KUKA KRL program: MyProgram_005().src

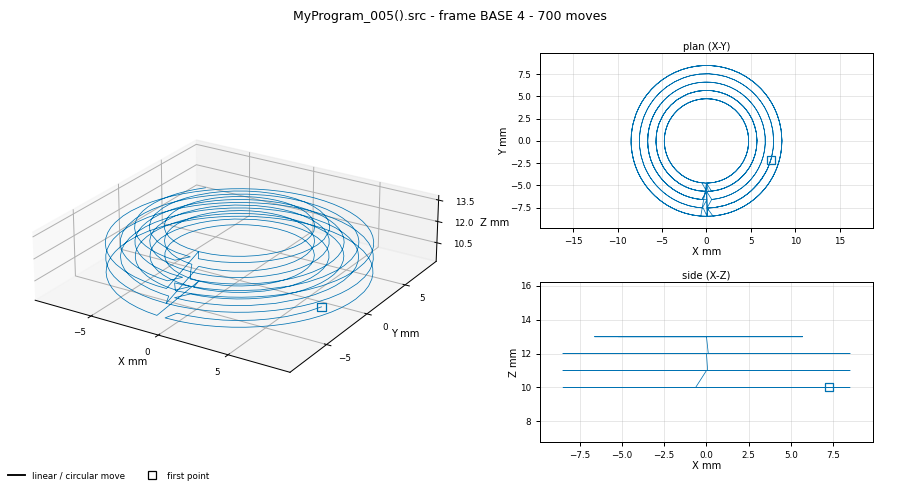
[picture p0: tool path of MyProgram_005().src in frame BASE 4, 700 of 700 moves have a stored position in this frame; points joined in program order, loops and branches not executed]
&ACCESS RVP
&REL 1
&PARAM TEMPLATE = C:\KRC\Roboter\Template\vorgabe
&PARAM EDITMASK = *
DEF MyProgram_005()
; ---- Setting reference (Base) ----
$BASE = BASE_DATA[4]

; --------------------------
; ---- Setting tool (TCP) ----
$TOOL = TOOL_DATA[3]
; --------------------------

$VEL.CP = VEL_APROX_PRINT
Startdeposition()
$VEL.CP = VEL_PRINT
LIN {X 7.2514,Y -2.1135,Z 10,A -2.621,B 0,C 0,E1 0.1598,E2 90.0715} C_DIS
LIN {X 6.8282,Y -3.2375,Z 10,A -2.6842,B 0,C 0,E1 0.1598,E2 90.0713} C_DIS
LIN {X 6.1189,Y -4.4371,Z 10,A -2.7612,B 0,C 0,E1 0.1598,E2 90.0712} C_DIS
LIN {X 5.3653,Y -5.3155,Z 10,A -2.8264,B 0,C 0,E1 0.1598,E2 90.0714} C_DIS
LIN {X 4.7502,Y -5.8723,Z 10,A -2.8729,B 0,C 0,E1 0.1598,E2 90.0716} C_DIS
LIN {X 3.9033,Y -6.4707,Z 10,A -2.9293,B 0,C 0,E1 0.1598,E2 90.0715} C_DIS
LIN {X 3.121,Y -6.8841,Z 10,A -2.9756,B 0,C 0,E1 0.1598,E2 90.0715} C_DIS
LIN {X 2.0664,Y -7.2652,Z 10,A -3.0305,B 0,C 0,E1 0.1598,E2 90.0715} C_DIS
LIN {X 0.9259,Y -7.5003,Z 10,A -3.0823,B 0,C 0,E1 0.1598,E2 90.0715} C_DIS
LIN {X 0.2286,Y -7.5485,Z 10,A -3.11,B 0,C 0,E1 0.1598,E2 90.0715} C_DIS
LIN {X 0.2286,Y -7.5485,Z 10,A -3.11,B 0,C 0,E1 0.1598,E2 90.0715} C_DIS
Enddeposition()
LIN {X -0.0236,Y -8.4916,Z 10,A -3.1582,B 0,C 0,E1 0.1598,E2 90.0702} C_DIS
Startdeposition()
$VEL.CP = VEL_PRINT
LIN {X 0.9995,Y -8.4285,Z 10,A -3.1191,B 0,C 0,E1 0.1598,E2 90.0714} C_DIS
LIN {X 1.8081,Y -8.2918,Z 10,A -3.0837,B 0,C 0,E1 0.1598,E2 90.0714} C_DIS
LIN {X 2.5999,Y -8.0782,Z 10,A -3.0456,B 0,C 0,E1 0.1598,E2 90.0714} C_DIS
LIN {X 3.3672,Y -7.789,Z 10,A -3.0052,B 0,C 0,E1 0.1598,E2 90.0715} C_DIS
LIN {X 4.1031,Y -7.4274,Z 10,A -2.9629,B 0,C 0,E1 0.1598,E2 90.0715} C_DIS
LIN {X 4.8011,Y -6.9971,Z 10,A -2.919,B 0,C 0,E1 0.1598,E2 90.0715} C_DIS
LIN {X 5.4543,Y -6.5014,Z 10,A -2.8739,B 0,C 0,E1 0.1598,E2 90.0716} C_DIS
LIN {X 6.0566,Y -5.9451,Z 10,A -2.8282,B 0,C 0,E1 0.1598,E2 90.0716} C_DIS
LIN {X 6.6023,Y -5.3331,Z 10,A -2.7821,B 0,C 0,E1 0.1598,E2 90.0716} C_DIS
LIN {X 7.0858,Y -4.6709,Z 10,A -2.7362,B 0,C 0,E1 0.1598,E2 90.0716} C_DIS
LIN {X 7.5037,Y -3.9655,Z 10,A -2.6908,B 0,C 0,E1 0.1598,E2 90.0717} C_DIS
LIN {X 7.8515,Y -3.2229,Z 10,A -2.6464,B 0,C 0,E1 0.1598,E2 90.0717} C_DIS
LIN {X 8.1262,Y -2.4503,Z 10,A -2.6035,B 0,C 0,E1 0.1598,E2 90.0717} C_DIS
LIN {X 8.3251,Y -1.6548,Z 10,A -2.5623,B 0,C 0,E1 0.1598,E2 90.0718} C_DIS
LIN {X 8.4456,Y -0.8436,Z 10,A -2.5234,B 0,C 0,E1 0.1598,E2 90.0718} C_DIS
LIN {X 8.4871,Y -0.0246,Z 10,A -2.4871,B 0,C 0,E1 0.1598,E2 90.0718} C_DIS
LIN {X 8.4059,Y 1.2036,Z 10,A -2.4375,B 0,C 0,E1 0.1598,E2 90.0715} C_DIS
LIN {X 8.2317,Y 2.0804,Z 10,A -2.4069,B 0,C 0,E1 0.1598,E2 90.0718} C_DIS
LIN {X 7.9103,Y 3.0772,Z 10,A -2.3765,B 0,C 0,E1 0.1598,E2 90.0718} C_DIS
LIN {X 7.5683,Y 3.8421,Z 10,A -2.3568,B 0,C 0,E1 0.1598,E2 90.0721} C_DIS
LIN {X 7.1528,Y 4.5697,Z 10,A -2.3413,B 0,C 0,E1 0.1598,E2 90.0721} C_DIS
LIN {X 6.6677,Y 5.253,Z 10,A -2.3302,B 0,C 0,E1 0.1598,E2 90.0721} C_DIS
LIN {X 6.1178,Y 5.8852,Z 10,A -2.3238,B 0,C 0,E1 0.1598,E2 90.0722} C_DIS
LIN {X 5.3488,Y 6.5961,Z 10,A -2.3219,B 0,C 0,E1 0.1598,E2 90.0722} C_DIS
LIN {X 4.4236,Y 7.2439,Z 10,A -2.3287,B 0,C 0,E1 0.1598,E2 90.0722} C_DIS
LIN {X 3.6959,Y 7.6405,Z 10,A -2.339,B 0,C 0,E1 0.1598,E2 90.0723} C_DIS
LIN {X 2.9332,Y 7.9646,Z 10,A -2.3535,B 0,C 0,E1 0.1598,E2 90.0723} C_DIS
LIN {X 2.1425,Y 8.213,Z 10,A -2.3722,B 0,C 0,E1 0.1598,E2 90.0723} C_DIS
LIN {X 1.3315,Y 8.3834,Z 10,A -2.395,B 0,C 0,E1 0.1598,E2 90.0723} C_DIS
LIN {X 0.5076,Y 8.4735,Z 10,A -2.4216,B 0,C 0,E1 0.1598,E2 90.0723} C_DIS
LIN {X -0.3211,Y 8.4813,Z 10,A -2.4519,B 0,C 0,E1 0.1598,E2 90.0723} C_DIS
LIN {X -1.1466,Y 8.4087,Z 10,A -2.4855,B 0,C 0,E1 0.1598,E2 90.0723} C_DIS
LIN {X -1.9613,Y 8.2569,Z 10,A -2.522,B 0,C 0,E1 0.1598,E2 90.0723} C_DIS
LIN {X -2.7572,Y 8.026,Z 10,A -2.5611,B 0,C 0,E1 0.1598,E2 90.0721} C_DIS
LIN {X -3.527,Y 7.7188,Z 10,A -2.6024,B 0,C 0,E1 0.1598,E2 90.0721} C_DIS
LIN {X -4.2632,Y 7.3382,Z 10,A -2.6456,B 0,C 0,E1 0.1598,E2 90.072} C_DIS
LIN {X -4.9588,Y 6.8878,Z 10,A -2.6902,B 0,C 0,E1 0.1598,E2 90.0719} C_DIS
LIN {X -5.607,Y 6.3713,Z 10,A -2.7358,B 0,C 0,E1 0.1598,E2 90.0718} C_DIS
LIN {X -6.2028,Y 5.7951,Z 10,A -2.782,B 0,C 0,E1 0.1598,E2 90.0718} C_DIS
LIN {X -6.7386,Y 5.1628,Z 10,A -2.8283,B 0,C 0,E1 0.1598,E2 90.0716} C_DIS
LIN {X -7.2097,Y 4.4809,Z 10,A -2.8743,B 0,C 0,E1 0.1598,E2 90.0716} C_DIS
LIN {X -7.6121,Y 3.7563,Z 10,A -2.9196,B 0,C 0,E1 0.1598,E2 90.0714} C_DIS
LIN {X -7.9422,Y 2.996,Z 10,A -2.9637,B 0,C 0,E1 0.1598,E2 90.0714} C_DIS
LIN {X -8.291,Y 1.8311,Z 10,A -3.0252,B 0,C 0,E1 0.1598,E2 90.0709} C_DIS
LIN {X -8.4593,Y 0.7466,Z 10,A -3.077,B 0,C 0,E1 0.1598,E2 90.0709} C_DIS
LIN {X -8.4789,Y -0.3697,Z 10,A -3.1246,B 0,C 0,E1 0.1598,E2 90.0707} C_DIS
LIN {X -8.4027,Y -1.1872,Z 10,A -3.1566,B 0,C 0,E1 0.1598,E2 90.071} C_DIS
LIN {X -8.2484,Y -1.9937,Z 10,A -3.1848,B 0,C 0,E1 0.1598,E2 90.071} C_DIS
LIN {X -8.0171,Y -2.7815,Z 10,A -3.2095,B 0,C 0,E1 0.1598,E2 90.071} C_DIS
LIN {X -7.7109,Y -3.5434,Z 10,A -3.2304,B 0,C 0,E1 0.1598,E2 90.071} C_DIS
LIN {X -7.3327,Y -4.2722,Z 10,A -3.2472,B 0,C 0,E1 0.1598,E2 90.071} C_DIS
LIN {X -6.8859,Y -4.9612,Z 10,A -3.2599,B 0,C 0,E1 0.1598,E2 90.071} C_DIS
LIN {X -6.3741,Y -5.6034,Z 10,A -3.2682,B 0,C 0,E1 0.1598,E2 90.071} C_DIS
LIN {X -5.8014,Y -6.1919,Z 10,A -3.2721,B 0,C 0,E1 0.1598,E2 90.071} C_DIS
LIN {X -5.176,Y -6.7238,Z 10,A -3.2716,B 0,C 0,E1 0.1598,E2 90.071} C_DIS
LIN {X -4.5041,Y -7.1958,Z 10,A -3.2669,B 0,C 0,E1 0.1598,E2 90.071} C_DIS
LIN {X -3.7871,Y -7.5963,Z 10,A -3.2576,B 0,C 0,E1 0.1598,E2 90.0711} C_DIS
LIN {X -3.0353,Y -7.9267,Z 10,A -3.244,B 0,C 0,E1 0.1598,E2 90.0711} C_DIS
LIN {X -2.2551,Y -8.1827,Z 10,A -3.2263,B 0,C 0,E1 0.1598,E2 90.0712} C_DIS
LIN {X -1.4539,Y -8.3624,Z 10,A -3.2045,B 0,C 0,E1 0.1598,E2 90.0712} C_DIS
LIN {X -0.639,Y -8.4635,Z 10,A -3.179,B 0,C 0,E1 0.1598,E2 90.0713} C_DIS
LIN {X -0.639,Y -8.4635,Z 10,A -3.179,B 0,C 0,E1 0.1598,E2 90.0713} C_DIS
Enddeposition()
LIN {X 0.0003,Y -4.7568,Z 11,A -2.9833,B 0,C 0,E1 0.1598,E2 90.0604} C_DIS
Startdeposition()
$VEL.CP = VEL_PRINT
LIN {X 0.0003,Y -4.7568,Z 11,A -2.9889,B 0,C 0,E1 0.1598,E2 90.0661} C_DIS
LIN {X -0.8726,Y -4.6702,Z 11,A -3.0221,B 0,C 0,E1 0.1598,E2 90.0709} C_DIS
LIN {X -1.5511,Y -4.491,Z 11,A -3.0401,B 0,C 0,E1 0.1598,E2 90.0715} C_DIS
LIN {X -2.1956,Y -4.2133,Z 11,A -3.052,B 0,C 0,E1 0.1598,E2 90.0715} C_DIS
LIN {X -2.7922,Y -3.844,Z 11,A -3.0583,B 0,C 0,E1 0.1598,E2 90.0715} C_DIS
LIN {X -3.3272,Y -3.3898,Z 11,A -3.0587,B 0,C 0,E1 0.1598,E2 90.0714} C_DIS
LIN {X -3.7898,Y -2.8623,Z 11,A -3.0534,B 0,C 0,E1 0.1598,E2 90.0714} C_DIS
LIN {X -4.1709,Y -2.2731,Z 11,A -3.0425,B 0,C 0,E1 0.1598,E2 90.0714} C_DIS
LIN {X -4.4614,Y -1.6344,Z 11,A -3.0262,B 0,C 0,E1 0.1598,E2 90.0714} C_DIS
LIN {X -4.6534,Y -0.9593,Z 11,A -3.0047,B 0,C 0,E1 0.1598,E2 90.0714} C_DIS
LIN {X -4.7423,Y -0.2633,Z 11,A -2.9786,B 0,C 0,E1 0.1598,E2 90.0714} C_DIS
LIN {X -4.731,Y 0.4382,Z 11,A -2.9486,B 0,C 0,E1 0.1598,E2 90.0714} C_DIS
LIN {X -4.6153,Y 1.1305,Z 11,A -2.9152,B 0,C 0,E1 0.1598,E2 90.0714} C_DIS
LIN {X -4.3961,Y 1.7972,Z 11,A -2.879,B 0,C 0,E1 0.1598,E2 90.0715} C_DIS
LIN {X -4.0858,Y 2.4265,Z 11,A -2.8411,B 0,C 0,E1 0.1598,E2 90.0715} C_DIS
LIN {X -3.6841,Y 3.0021,Z 11,A -2.802,B 0,C 0,E1 0.1598,E2 90.0717} C_DIS
LIN {X -3.2012,Y 3.5114,Z 11,A -2.7628,B 0,C 0,E1 0.1598,E2 90.0717} C_DIS
LIN {X -2.6493,Y 3.9451,Z 11,A -2.7242,B 0,C 0,E1 0.1598,E2 90.0719} C_DIS
LIN {X -2.0393,Y 4.2923,Z 11,A -2.6871,B 0,C 0,E1 0.1598,E2 90.0719} C_DIS
LIN {X -1.3842,Y 4.5438,Z 11,A -2.6524,B 0,C 0,E1 0.1598,E2 90.072} C_DIS
LIN {X -0.6998,Y 4.6984,Z 11,A -2.6206,B 0,C 0,E1 0.1598,E2 90.072} C_DIS
LIN {X -0.0003,Y 4.75,Z 11,A -2.5927,B 0,C 0,E1 0.1598,E2 90.0721} C_DIS
LIN {X 0.6994,Y 4.6987,Z 11,A -2.569,B 0,C 0,E1 0.1598,E2 90.0721} C_DIS
LIN {X 1.3838,Y 4.5442,Z 11,A -2.5503,B 0,C 0,E1 0.1598,E2 90.0721} C_DIS
LIN {X 2.039,Y 4.2925,Z 11,A -2.5368,B 0,C 0,E1 0.1598,E2 90.0721} C_DIS
LIN {X 2.6481,Y 3.9439,Z 11,A -2.529,B 0,C 0,E1 0.1598,E2 90.0721} C_DIS
LIN {X 3.1999,Y 3.5104,Z 11,A -2.527,B 0,C 0,E1 0.1598,E2 90.0721} C_DIS
LIN {X 3.6819,Y 3.0005,Z 11,A -2.5308,B 0,C 0,E1 0.1598,E2 90.0721} C_DIS
LIN {X 4.0854,Y 2.4265,Z 11,A -2.5402,B 0,C 0,E1 0.1598,E2 90.072} C_DIS
LIN {X 4.3971,Y 1.7978,Z 11,A -2.5553,B 0,C 0,E1 0.1598,E2 90.072} C_DIS
LIN {X 4.6137,Y 1.1305,Z 11,A -2.5756,B 0,C 0,E1 0.1598,E2 90.0719} C_DIS
LIN {X 4.7302,Y 0.4386,Z 11,A -2.6006,B 0,C 0,E1 0.1598,E2 90.0719} C_DIS
LIN {X 4.7449,Y -0.2631,Z 11,A -2.6298,B 0,C 0,E1 0.1598,E2 90.0718} C_DIS
LIN {X 4.6542,Y -0.959,Z 11,A -2.6627,B 0,C 0,E1 0.1598,E2 90.0718} C_DIS
LIN {X 4.4618,Y -1.634,Z 11,A -2.6984,B 0,C 0,E1 0.1598,E2 90.0718} C_DIS
LIN {X 4.1713,Y -2.2727,Z 11,A -2.7362,B 0,C 0,E1 0.1598,E2 90.0718} C_DIS
LIN {X 3.7907,Y -2.8621,Z 11,A -2.7752,B 0,C 0,E1 0.1598,E2 90.0717} C_DIS
LIN {X 3.2003,Y -3.51,Z 11,A -2.8243,B 0,C 0,E1 0.1598,E2 90.0717} C_DIS
LIN {X 2.648,Y -3.9429,Z 11,A -2.8631,B 0,C 0,E1 0.1598,E2 90.0717} C_DIS
LIN {X 2.1966,Y -4.2139,Z 11,A -2.8912,B 0,C 0,E1 0.1598,E2 90.0717} C_DIS
LIN {X 1.5512,Y -4.4896,Z 11,A -2.9266,B 0,C 0,E1 0.1598,E2 90.0717} C_DIS
LIN {X 0.8732,Y -4.6704,Z 11,A -2.9591,B 0,C 0,E1 0.1598,E2 90.0717} C_DIS
LIN {X 0.0003,Y -4.7568,Z 11,A -2.9948,B 0,C 0,E1 0.1598,E2 90.0716} C_DIS
Enddeposition()
LIN {X 0.0003,Y -4.7568,Z 11,A -2.9948,B 0,C 0,E1 0.1598,E2 90.0716} C_DIS
Startdeposition()
$VEL.CP = VEL_PRINT
LIN {X 0.2115,Y -5.6786,Z 11,A -3.0257,B 0,C 0,E1 0.1598,E2 90.071} C_DIS
LIN {X 1.0414,Y -5.5858,Z 11,A -2.9918,B 0,C 0,E1 0.1598,E2 90.0716} C_DIS
LIN {X 1.849,Y -5.3736,Z 11,A -2.9532,B 0,C 0,E1 0.1598,E2 90.0716} C_DIS
LIN {X 2.6171,Y -5.0456,Z 11,A -2.9111,B 0,C 0,E1 0.1598,E2 90.0716} C_DIS
LIN {X 3.3282,Y -4.6074,Z 11,A -2.8663,B 0,C 0,E1 0.1598,E2 90.0716} C_DIS
LIN {X 4.1901,Y -3.8495,Z 11,A -2.8024,B 0,C 0,E1 0.1598,E2 90.0716} C_DIS
LIN {X 4.8132,Y -3.0255,Z 11,A -2.7445,B 0,C 0,E1 0.1598,E2 90.0716} C_DIS
LIN {X 5.201,Y -2.2955,Z 11,A -2.6993,B 0,C 0,E1 0.1598,E2 90.0716} C_DIS
LIN {X 5.4794,Y -1.5173,Z 11,A -2.656,B 0,C 0,E1 0.1598,E2 90.0717} C_DIS
LIN {X 5.641,Y -0.7067,Z 11,A -2.6156,B 0,C 0,E1 0.1598,E2 90.0717} C_DIS
LIN {X 5.6825,Y 0.1187,Z 11,A -2.579,B 0,C 0,E1 0.1598,E2 90.0717} C_DIS
LIN {X 5.6056,Y 0.9414,Z 11,A -2.547,B 0,C 0,E1 0.1598,E2 90.0718} C_DIS
LIN {X 5.4111,Y 1.7446,Z 11,A -2.5201,B 0,C 0,E1 0.1598,E2 90.0718} C_DIS
LIN {X 5.1013,Y 2.5109,Z 11,A -2.499,B 0,C 0,E1 0.1598,E2 90.0719} C_DIS
LIN {X 4.6827,Y 3.2236,Z 11,A -2.4843,B 0,C 0,E1 0.1598,E2 90.0719} C_DIS
LIN {X 4.165,Y 3.8679,Z 11,A -2.4761,B 0,C 0,E1 0.1598,E2 90.072} C_DIS
LIN {X 3.5608,Y 4.4318,Z 11,A -2.4746,B 0,C 0,E1 0.1598,E2 90.072} C_DIS
LIN {X 2.8804,Y 4.9013,Z 11,A -2.4799,B 0,C 0,E1 0.1598,E2 90.0721} C_DIS
LIN {X 2.1391,Y 5.2669,Z 11,A -2.4918,B 0,C 0,E1 0.1598,E2 90.0721} C_DIS
LIN {X 1.3523,Y 5.5201,Z 11,A -2.5101,B 0,C 0,E1 0.1598,E2 90.0721} C_DIS
LIN {X 0.5378,Y 5.659,Z 11,A -2.5344,B 0,C 0,E1 0.1598,E2 90.0721} C_DIS
LIN {X -0.2883,Y 5.6764,Z 11,A -2.5641,B 0,C 0,E1 0.1598,E2 90.0721} C_DIS
LIN {X -1.1084,Y 5.5748,Z 11,A -2.5986,B 0,C 0,E1 0.1598,E2 90.0721} C_DIS
LIN {X -2.1006,Y 5.2877,Z 11,A -2.6473,B 0,C 0,E1 0.1598,E2 90.072} C_DIS
LIN {X -3.2896,Y 4.6422,Z 11,A -2.7182,B 0,C 0,E1 0.1598,E2 90.0717} C_DIS
LIN {X -3.9903,Y 4.0465,Z 11,A -2.7692,B 0,C 0,E1 0.1598,E2 90.0717} C_DIS
LIN {X -4.4802,Y 3.4976,Z 11,A -2.8104,B 0,C 0,E1 0.1598,E2 90.0717} C_DIS
LIN {X -4.8958,Y 2.8906,Z 11,A -2.8512,B 0,C 0,E1 0.1598,E2 90.0716} C_DIS
LIN {X -5.3507,Y 1.9338,Z 11,A -2.9081,B 0,C 0,E1 0.1598,E2 90.0713} C_DIS
LIN {X -5.5909,Y 1.0258,Z 11,A -2.9552,B 0,C 0,E1 0.1598,E2 90.0713} C_DIS
LIN {X -5.6775,Y 0.2794,Z 11,A -2.9899,B 0,C 0,E1 0.1598,E2 90.0713} C_DIS
LIN {X -5.6649,Y -0.4718,Z 11,A -3.0211,B 0,C 0,E1 0.1598,E2 90.0713} C_DIS
LIN {X -5.5534,Y -1.2149,Z 11,A -3.0484,B 0,C 0,E1 0.1598,E2 90.0713} C_DIS
LIN {X -5.3437,Y -1.9363,Z 11,A -3.0711,B 0,C 0,E1 0.1598,E2 90.0713} C_DIS
LIN {X -5.0406,Y -2.6238,Z 11,A -3.089,B 0,C 0,E1 0.1598,E2 90.0713} C_DIS
LIN {X -4.6521,Y -3.2668,Z 11,A -3.1019,B 0,C 0,E1 0.1598,E2 90.0713} C_DIS
LIN {X -4.1812,Y -3.8525,Z 11,A -3.1093,B 0,C 0,E1 0.1598,E2 90.0713} C_DIS
LIN {X -3.6366,Y -4.3703,Z 11,A -3.1112,B 0,C 0,E1 0.1598,E2 90.0713} C_DIS
LIN {X -3.0273,Y -4.8101,Z 11,A -3.1075,B 0,C 0,E1 0.1598,E2 90.0713} C_DIS
LIN {X -2.3672,Y -5.1692,Z 11,A -3.0985,B 0,C 0,E1 0.1598,E2 90.0713} C_DIS
LIN {X -1.6648,Y -5.4362,Z 11,A -3.084,B 0,C 0,E1 0.1598,E2 90.0714} C_DIS
LIN {X -0.933,Y -5.6073,Z 11,A -3.0644,B 0,C 0,E1 0.1598,E2 90.0714} C_DIS
LIN {X 0.0026,Y -5.6868,Z 11,A -3.0334,B 0,C 0,E1 0.1598,E2 90.0715} C_DIS
Enddeposition()
LIN {X 0.0026,Y -5.6868,Z 11,A -3.0334,B 0,C 0,E1 0.1598,E2 90.0715} C_DIS
Startdeposition()
$VEL.CP = VEL_PRINT
LIN {X -0.4949,Y -6.6014,Z 11,A -3.09,B 0,C 0,E1 0.1598,E2 90.0709} C_DIS
LIN {X -1.1902,Y -6.5105,Z 11,A -3.1122,B 0,C 0,E1 0.1598,E2 90.0714} C_DIS
LIN {X -1.8726,Y -6.3494,Z 11,A -3.1304,B 0,C 0,E1 0.1598,E2 90.0714} C_DIS
LIN {X -2.5337,Y -6.1155,Z 11,A -3.1448,B 0,C 0,E1 0.1598,E2 90.0714} C_DIS
LIN {X -3.1661,Y -5.8125,Z 11,A -3.1552,B 0,C 0,E1 0.1598,E2 90.0714} C_DIS
LIN {X -3.7646,Y -5.4468,Z 11,A -3.1616,B 0,C 0,E1 0.1598,E2 90.0713} C_DIS
LIN {X -4.3185,Y -5.0169,Z 11,A -3.1638,B 0,C 0,E1 0.1598,E2 90.0713} C_DIS
LIN {X -4.8238,Y -4.5307,Z 11,A -3.1618,B 0,C 0,E1 0.1598,E2 90.0713} C_DIS
LIN {X -5.2766,Y -3.9954,Z 11,A -3.1558,B 0,C 0,E1 0.1598,E2 90.0713} C_DIS
LIN {X -5.6699,Y -3.415,Z 11,A -3.1457,B 0,C 0,E1 0.1598,E2 90.0713} C_DIS
LIN {X -5.999,Y -2.7958,Z 11,A -3.1317,B 0,C 0,E1 0.1598,E2 90.0712} C_DIS
LIN {X -6.2622,Y -2.1459,Z 11,A -3.1139,B 0,C 0,E1 0.1598,E2 90.0712} C_DIS
LIN {X -6.4548,Y -1.4716,Z 11,A -3.0926,B 0,C 0,E1 0.1598,E2 90.0712} C_DIS
LIN {X -6.5732,Y -0.7805,Z 11,A -3.0678,B 0,C 0,E1 0.1598,E2 90.0712} C_DIS
LIN {X -6.6178,Y -0.0807,Z 11,A -3.0399,B 0,C 0,E1 0.1598,E2 90.0712} C_DIS
LIN {X -6.5916,Y 0.62,Z 11,A -3.0094,B 0,C 0,E1 0.1598,E2 90.0713} C_DIS
LIN {X -6.4894,Y 1.3139,Z 11,A -2.9765,B 0,C 0,E1 0.1598,E2 90.0713} C_DIS
LIN {X -6.3129,Y 1.9925,Z 11,A -2.9414,B 0,C 0,E1 0.1598,E2 90.0714} C_DIS
LIN {X -6.0681,Y 2.6497,Z 11,A -2.9047,B 0,C 0,E1 0.1598,E2 90.0714} C_DIS
LIN {X -5.7534,Y 3.2763,Z 11,A -2.8667,B 0,C 0,E1 0.1598,E2 90.0716} C_DIS
LIN {X -5.3742,Y 3.8661,Z 11,A -2.8279,B 0,C 0,E1 0.1598,E2 90.0716} C_DIS
LIN {X -4.9335,Y 4.4116,Z 11,A -2.7888,B 0,C 0,E1 0.1598,E2 90.0717} C_DIS
LIN {X -4.4407,Y 4.9103,Z 11,A -2.7496,B 0,C 0,E1 0.1598,E2 90.0717} C_DIS
LIN {X -3.8964,Y 5.3524,Z 11,A -2.7109,B 0,C 0,E1 0.1598,E2 90.0719} C_DIS
LIN {X -3.3078,Y 5.7338,Z 11,A -2.6732,B 0,C 0,E1 0.1598,E2 90.0719} C_DIS
LIN {X -2.6834,Y 6.0528,Z 11,A -2.6367,B 0,C 0,E1 0.1598,E2 90.072} C_DIS
LIN {X -2.0284,Y 6.3032,Z 11,A -2.602,B 0,C 0,E1 0.1598,E2 90.072} C_DIS
LIN {X -1.3505,Y 6.4829,Z 11,A -2.5694,B 0,C 0,E1 0.1598,E2 90.0721} C_DIS
LIN {X -0.6569,Y 6.5864,Z 11,A -2.5395,B 0,C 0,E1 0.1598,E2 90.0721} C_DIS
LIN {X 0.0435,Y 6.6177,Z 11,A -2.5123,B 0,C 0,E1 0.1598,E2 90.0722} C_DIS
LIN {X 0.7435,Y 6.5781,Z 11,A -2.4881,B 0,C 0,E1 0.1598,E2 90.0722} C_DIS
LIN {X 1.4351,Y 6.4616,Z 11,A -2.4675,B 0,C 0,E1 0.1598,E2 90.0722} C_DIS
LIN {X 2.1108,Y 6.2745,Z 11,A -2.4505,B 0,C 0,E1 0.1598,E2 90.0722} C_DIS
LIN {X 2.7627,Y 6.0158,Z 11,A -2.4374,B 0,C 0,E1 0.1598,E2 90.0722} C_DIS
LIN {X 3.3832,Y 5.6892,Z 11,A -2.4283,B 0,C 0,E1 0.1598,E2 90.0722} C_DIS
LIN {X 3.966,Y 5.2993,Z 11,A -2.4232,B 0,C 0,E1 0.1598,E2 90.0722} C_DIS
LIN {X 4.6345,Y 4.7322,Z 11,A -2.4225,B 0,C 0,E1 0.1598,E2 90.0722} C_DIS
LIN {X 5.3297,Y 3.9254,Z 11,A -2.4308,B 0,C 0,E1 0.1598,E2 90.0719} C_DIS
LIN {X 5.7333,Y 3.3083,Z 11,A -2.4423,B 0,C 0,E1 0.1598,E2 90.0721} C_DIS
LIN {X 6.0651,Y 2.65,Z 11,A -2.4579,B 0,C 0,E1 0.1598,E2 90.0721} C_DIS
LIN {X 6.3215,Y 1.9587,Z 11,A -2.4778,B 0,C 0,E1 0.1598,E2 90.072} C_DIS
LIN {X 6.5003,Y 1.2436,Z 11,A -2.5015,B 0,C 0,E1 0.1598,E2 90.072} C_DIS
LIN {X 6.6002,Y 0.513,Z 11,A -2.5288,B 0,C 0,E1 0.1598,E2 90.072} C_DIS
LIN {X 6.6143,Y -0.2241,Z 11,A -2.5596,B 0,C 0,E1 0.1598,E2 90.0719} C_DIS
LIN {X 6.5512,Y -0.9586,Z 11,A -2.5931,B 0,C 0,E1 0.1598,E2 90.0719} C_DIS
LIN {X 6.4028,Y -1.6809,Z 11,A -2.6292,B 0,C 0,E1 0.1598,E2 90.0718} C_DIS
LIN {X 6.1763,Y -2.3825,Z 11,A -2.6673,B 0,C 0,E1 0.1598,E2 90.0718} C_DIS
LIN {X 5.8721,Y -3.0543,Z 11,A -2.707,B 0,C 0,E1 0.1598,E2 90.0718} C_DIS
LIN {X 5.4976,Y -3.6893,Z 11,A -2.7478,B 0,C 0,E1 0.1598,E2 90.0718} C_DIS
LIN {X 5.0529,Y -4.2774,Z 11,A -2.7891,B 0,C 0,E1 0.1598,E2 90.0717} C_DIS
LIN {X 4.5453,Y -4.8123,Z 11,A -2.8305,B 0,C 0,E1 0.1598,E2 90.0717} C_DIS
LIN {X 3.9811,Y -5.287,Z 11,A -2.8714,B 0,C 0,E1 0.1598,E2 90.0717} C_DIS
LIN {X 3.3686,Y -5.6973,Z 11,A -2.9113,B 0,C 0,E1 0.1598,E2 90.0717} C_DIS
LIN {X 2.7135,Y -6.0353,Z 11,A -2.9497,B 0,C 0,E1 0.1598,E2 90.0716} C_DIS
LIN {X 2.0261,Y -6.3017,Z 11,A -2.9862,B 0,C 0,E1 0.1598,E2 90.0716} C_DIS
LIN {X 1.3132,Y -6.49,Z 11,A -3.0204,B 0,C 0,E1 0.1598,E2 90.0716} C_DIS
LIN {X 0.5832,Y -6.5943,Z 11,A -3.0516,B 0,C 0,E1 0.1598,E2 90.0716} C_DIS
LIN {X 0.5832,Y -6.5943,Z 11,A -3.0516,B 0,C 0,E1 0.1598,E2 90.0716} C_DIS
Enddeposition()
LIN {X 0.0612,Y -7.5554,Z 11,A -3.1105,B 0,C 0,E1 0.1598,E2 90.0703} C_DIS
Startdeposition()
$VEL.CP = VEL_PRINT
LIN {X 0.9096,Y -7.5021,Z 11,A -3.0782,B 0,C 0,E1 0.1598,E2 90.0714} C_DIS
LIN {X 2.0698,Y -7.2637,Z 11,A -3.0256,B 0,C 0,E1 0.1598,E2 90.0715} C_DIS
LIN {X 3.159,Y -6.8663,Z 11,A -2.9687,B 0,C 0,E1 0.1598,E2 90.0715} C_DIS
LIN {X 3.97,Y -6.424,Z 11,A -2.9202,B 0,C 0,E1 0.1598,E2 90.0715} C_DIS
LIN {X 4.5787,Y -6.0051,Z 11,A -2.8801,B 0,C 0,E1 0.1598,E2 90.0716} C_DIS
LIN {X 5.6784,Y -4.9864,Z 11,A -2.7959,B 0,C 0,E1 0.1598,E2 90.0712} C_DIS
LIN {X 6.6606,Y -3.5697,Z 11,A -2.6993,B 0,C 0,E1 0.1598,E2 90.071} C_DIS
LIN {X 7.0779,Y -2.6472,Z 11,A -2.6453,B 0,C 0,E1 0.1598,E2 90.0716} C_DIS
LIN {X 7.3848,Y -1.592,Z 11,A -2.589,B 0,C 0,E1 0.1598,E2 90.0716} C_DIS
LIN {X 7.5054,Y -0.8566,Z 11,A -2.5537,B 0,C 0,E1 0.1598,E2 90.0719} C_DIS
LIN {X 7.557,Y 0.0734,Z 11,A -2.512,B 0,C 0,E1 0.1598,E2 90.0717} C_DIS
LIN {X 7.4618,Y 1.1945,Z 11,A -2.4678,B 0,C 0,E1 0.1598,E2 90.0717} C_DIS
LIN {X 7.2396,Y 2.1679,Z 11,A -2.4348,B 0,C 0,E1 0.1598,E2 90.0717} C_DIS
LIN {X 6.907,Y 3.0553,Z 11,A -2.4095,B 0,C 0,E1 0.1598,E2 90.0719} C_DIS
LIN {X 6.5658,Y 3.7322,Z 11,A -2.3935,B 0,C 0,E1 0.1598,E2 90.0721} C_DIS
LIN {X 6.1589,Y 4.3719,Z 11,A -2.3814,B 0,C 0,E1 0.1598,E2 90.0721} C_DIS
LIN {X 5.6894,Y 4.9671,Z 11,A -2.3736,B 0,C 0,E1 0.1598,E2 90.0721} C_DIS
LIN {X 5.1623,Y 5.5119,Z 11,A -2.3699,B 0,C 0,E1 0.1598,E2 90.0722} C_DIS
LIN {X 4.5834,Y 6.0012,Z 11,A -2.3706,B 0,C 0,E1 0.1598,E2 90.0722} C_DIS
LIN {X 3.9597,Y 6.4322,Z 11,A -2.3754,B 0,C 0,E1 0.1598,E2 90.0722} C_DIS
LIN {X 3.1257,Y 6.882,Z 11,A -2.3871,B 0,C 0,E1 0.1598,E2 90.0722} C_DIS
LIN {X 2.194,Y 7.2314,Z 11,A -2.4068,B 0,C 0,E1 0.1598,E2 90.0722} C_DIS
LIN {X 0.9897,Y 7.4881,Z 11,A -2.4405,B 0,C 0,E1 0.1598,E2 90.0722} C_DIS
LIN {X 0.239,Y 7.5535,Z 11,A -2.4655,B 0,C 0,E1 0.1598,E2 90.0722} C_DIS
LIN {X -0.7725,Y 7.5177,Z 11,A -2.5043,B 0,C 0,E1 0.1598,E2 90.0722} C_DIS
LIN {X -1.736,Y 7.3564,Z 11,A -2.5467,B 0,C 0,E1 0.1598,E2 90.0722} C_DIS
LIN {X -2.7886,Y 7.0254,Z 11,A -2.5995,B 0,C 0,E1 0.1598,E2 90.0721} C_DIS
LIN {X -3.6563,Y 6.6078,Z 11,A -2.6491,B 0,C 0,E1 0.1598,E2 90.072} C_DIS
LIN {X -4.4708,Y 6.0944,Z 11,A -2.7007,B 0,C 0,E1 0.1598,E2 90.0718} C_DIS
LIN {X -5.3112,Y 5.37,Z 11,A -2.762,B 0,C 0,E1 0.1598,E2 90.0716} C_DIS
LIN {X -5.8426,Y 4.7877,Z 11,A -2.8062,B 0,C 0,E1 0.1598,E2 90.0716} C_DIS
LIN {X -6.3083,Y 4.1518,Z 11,A -2.8501,B 0,C 0,E1 0.1598,E2 90.0716} C_DIS
LIN {X -6.708,Y 3.4725,Z 11,A -2.8934,B 0,C 0,E1 0.1598,E2 90.0715} C_DIS
LIN {X -7.1059,Y 2.571,Z 11,A -2.9458,B 0,C 0,E1 0.1598,E2 90.0712} C_DIS
LIN {X -7.4227,Y 1.3948,Z 11,A -3.0067,B 0,C 0,E1 0.1598,E2 90.0708} C_DIS
LIN {X -7.5368,Y 0.5156,Z 11,A -3.0482,B 0,C 0,E1 0.1598,E2 90.0711} C_DIS
LIN {X -7.5341,Y -0.5927,Z 11,A -3.0945,B 0,C 0,E1 0.1598,E2 90.0707} C_DIS
LIN {X -7.3917,Y -1.5706,Z 11,A -3.1306,B 0,C 0,E1 0.1598,E2 90.0709} C_DIS
LIN {X -7.0689,Y -2.6624,Z 11,A -3.1646,B 0,C 0,E1 0.1598,E2 90.0707} C_DIS
LIN {X -6.7741,Y -3.3489,Z 11,A -3.183,B 0,C 0,E1 0.1598,E2 90.071} C_DIS
LIN {X -6.2739,Y -4.2128,Z 11,A -3.201,B 0,C 0,E1 0.1598,E2 90.071} C_DIS
LIN {X -5.5619,Y -5.1165,Z 11,A -3.213,B 0,C 0,E1 0.1598,E2 90.0709} C_DIS
LIN {X -4.8434,Y -5.795,Z 11,A -3.2154,B 0,C 0,E1 0.1598,E2 90.0711} C_DIS
LIN {X -4.2115,Y -6.27,Z 11,A -3.2124,B 0,C 0,E1 0.1598,E2 90.0711} C_DIS
LIN {X -3.5333,Y -6.6762,Z 11,A -3.2047,B 0,C 0,E1 0.1598,E2 90.0712} C_DIS
LIN {X -2.8161,Y -7.009,Z 11,A -3.1925,B 0,C 0,E1 0.1598,E2 90.0712} C_DIS
LIN {X -1.8779,Y -7.3197,Z 11,A -3.1713,B 0,C 0,E1 0.1598,E2 90.0712} C_DIS
LIN {X -0.9529,Y -7.4938,Z 11,A -3.1448,B 0,C 0,E1 0.1598,E2 90.0714} C_DIS
LIN {X -0.3743,Y -7.5452,Z 11,A -3.1257,B 0,C 0,E1 0.1598,E2 90.0714} C_DIS
LIN {X -0.3743,Y -7.5452,Z 11,A -3.1257,B 0,C 0,E1 0.1598,E2 90.0714} C_DIS
Enddeposition()
LIN {X 0.0683,Y -8.4871,Z 11,A -3.1485,B 0,C 0,E1 0.1598,E2 90.0702} C_DIS
Startdeposition()
$VEL.CP = VEL_PRINT
LIN {X -0.9758,Y -8.4305,Z 11,A -3.1854,B 0,C 0,E1 0.1598,E2 90.0713} C_DIS
LIN {X -1.8014,Y -8.2948,Z 11,A -3.21,B 0,C 0,E1 0.1598,E2 90.0713} C_DIS
LIN {X -2.6094,Y -8.0774,Z 11,A -3.2304,B 0,C 0,E1 0.1598,E2 90.0713} C_DIS
LIN {X -3.3919,Y -7.781,Z 11,A -3.2465,B 0,C 0,E1 0.1598,E2 90.0712} C_DIS
LIN {X -4.1418,Y -7.4099,Z 11,A -3.2583,B 0,C 0,E1 0.1598,E2 90.0712} C_DIS
LIN {X -4.8515,Y -6.9664,Z 11,A -3.2656,B 0,C 0,E1 0.1598,E2 90.0712} C_DIS
LIN {X -5.5138,Y -6.455,Z 11,A -3.2682,B 0,C 0,E1 0.1598,E2 90.0711} C_DIS
LIN {X -6.1215,Y -5.8798,Z 11,A -3.2662,B 0,C 0,E1 0.1598,E2 90.0711} C_DIS
LIN {X -6.6696,Y -5.2475,Z 11,A -3.2596,B 0,C 0,E1 0.1598,E2 90.0711} C_DIS
LIN {X -7.1551,Y -4.566,Z 11,A -3.2486,B 0,C 0,E1 0.1598,E2 90.071} C_DIS
LIN {X -7.5698,Y -3.8392,Z 11,A -3.2332,B 0,C 0,E1 0.1598,E2 90.071} C_DIS
LIN {X -7.9111,Y -3.0751,Z 11,A -3.2135,B 0,C 0,E1 0.1598,E2 90.071} C_DIS
LIN {X -8.1756,Y -2.2812,Z 11,A -3.1898,B 0,C 0,E1 0.1598,E2 90.071} C_DIS
LIN {X -8.397,Y -1.2589,Z 11,A -3.1546,B 0,C 0,E1 0.1598,E2 90.0707} C_DIS
LIN {X -8.4874,Y -0.2374,Z 11,A -3.115,B 0,C 0,E1 0.1598,E2 90.0709} C_DIS
LIN {X -8.4598,Y 0.7402,Z 11,A -3.0728,B 0,C 0,E1 0.1598,E2 90.0709} C_DIS
LIN {X -8.291,Y 1.8311,Z 11,A -3.0206,B 0,C 0,E1 0.1598,E2 90.0709} C_DIS
LIN {X -7.9448,Y 2.9894,Z 11,A -2.9591,B 0,C 0,E1 0.1598,E2 90.0709} C_DIS
LIN {X -7.6152,Y 3.7501,Z 11,A -2.9153,B 0,C 0,E1 0.1598,E2 90.0714} C_DIS
LIN {X -7.2133,Y 4.4752,Z 11,A -2.87,B 0,C 0,E1 0.1598,E2 90.0714} C_DIS
LIN {X -6.7426,Y 5.1576,Z 11,A -2.824,B 0,C 0,E1 0.1598,E2 90.0716} C_DIS
LIN {X -6.2071,Y 5.7903,Z 11,A -2.7776,B 0,C 0,E1 0.1598,E2 90.0716} C_DIS
LIN {X -5.6121,Y 6.3676,Z 11,A -2.7314,B 0,C 0,E1 0.1598,E2 90.0718} C_DIS
LIN {X -4.9638,Y 6.8842,Z 11,A -2.6858,B 0,C 0,E1 0.1598,E2 90.0718} C_DIS
LIN {X -4.2682,Y 7.3352,Z 11,A -2.6412,B 0,C 0,E1 0.1598,E2 90.072} C_DIS
LIN {X -3.5321,Y 7.7164,Z 11,A -2.598,B 0,C 0,E1 0.1598,E2 90.072} C_DIS
LIN {X -2.7624,Y 8.0241,Z 11,A -2.5566,B 0,C 0,E1 0.1598,E2 90.0721} C_DIS
LIN {X -1.9665,Y 8.2556,Z 11,A -2.5175,B 0,C 0,E1 0.1598,E2 90.0721} C_DIS
LIN {X -1.1517,Y 8.408,Z 11,A -2.481,B 0,C 0,E1 0.1598,E2 90.0723} C_DIS
LIN {X -0.3261,Y 8.481,Z 11,A -2.4474,B 0,C 0,E1 0.1598,E2 90.0723} C_DIS
LIN {X 0.5028,Y 8.4738,Z 11,A -2.4171,B 0,C 0,E1 0.1598,E2 90.0723} C_DIS
LIN {X 1.3269,Y 8.3843,Z 11,A -2.3904,B 0,C 0,E1 0.1598,E2 90.0723} C_DIS
LIN {X 2.1382,Y 8.2143,Z 11,A -2.3676,B 0,C 0,E1 0.1598,E2 90.0723} C_DIS
LIN {X 2.9292,Y 7.9662,Z 11,A -2.3489,B 0,C 0,E1 0.1598,E2 90.0723} C_DIS
LIN {X 3.6923,Y 7.6424,Z 11,A -2.3344,B 0,C 0,E1 0.1598,E2 90.0723} C_DIS
LIN {X 4.4202,Y 7.246,Z 11,A -2.3242,B 0,C 0,E1 0.1598,E2 90.0723} C_DIS
LIN {X 5.345,Y 6.5991,Z 11,A -2.3173,B 0,C 0,E1 0.1598,E2 90.0723} C_DIS
LIN {X 6.1206,Y 5.8817,Z 11,A -2.3191,B 0,C 0,E1 0.1598,E2 90.0722} C_DIS
LIN {X 6.6747,Y 5.2434,Z 11,A -2.3257,B 0,C 0,E1 0.1598,E2 90.0722} C_DIS
LIN {X 7.1626,Y 4.5532,Z 11,A -2.3369,B 0,C 0,E1 0.1598,E2 90.0722} C_DIS
LIN {X 7.5797,Y 3.818,Z 11,A -2.3527,B 0,C 0,E1 0.1598,E2 90.0722} C_DIS
LIN {X 7.9217,Y 3.0451,Z 11,A -2.3729,B 0,C 0,E1 0.1598,E2 90.0721} C_DIS
LIN {X 8.1853,Y 2.242,Z 11,A -2.3972,B 0,C 0,E1 0.1598,E2 90.0721} C_DIS
LIN {X 8.4051,Y 1.2086,Z 11,A -2.4327,B 0,C 0,E1 0.1598,E2 90.0716} C_DIS
LIN {X 8.4904,Y 0.1014,Z 11,A -2.4766,B 0,C 0,E1 0.1598,E2 90.0716} C_DIS
LIN {X 8.4408,Y -0.891,Z 11,A -2.5207,B 0,C 0,E1 0.1598,E2 90.0717} C_DIS
LIN {X 8.3214,Y -1.6769,Z 11,A -2.5587,B 0,C 0,E1 0.1598,E2 90.0718} C_DIS
LIN {X 8.0706,Y -2.6384,Z 11,A -2.6085,B 0,C 0,E1 0.1598,E2 90.0715} C_DIS
LIN {X 7.6152,Y -3.7515,Z 11,A -2.6725,B 0,C 0,E1 0.1598,E2 90.0713} C_DIS
LIN {X 7.2107,Y -4.4808,Z 11,A -2.7187,B 0,C 0,E1 0.1598,E2 90.0717} C_DIS
LIN {X 6.7362,Y -5.1668,Z 11,A -2.7653,B 0,C 0,E1 0.1598,E2 90.0717} C_DIS
LIN {X 6.1963,Y -5.8024,Z 11,A -2.8122,B 0,C 0,E1 0.1598,E2 90.0717} C_DIS
LIN {X 5.5962,Y -6.3816,Z 11,A -2.8588,B 0,C 0,E1 0.1598,E2 90.0716} C_DIS
LIN {X 4.9427,Y -6.8997,Z 11,A -2.9048,B 0,C 0,E1 0.1598,E2 90.0716} C_DIS
LIN {X 4.2415,Y -7.3512,Z 11,A -2.9498,B 0,C 0,E1 0.1598,E2 90.0716} C_DIS
LIN {X 3.4995,Y -7.7318,Z 11,A -2.9931,B 0,C 0,E1 0.1598,E2 90.0716} C_DIS
LIN {X 2.7238,Y -8.0379,Z 11,A -3.0346,B 0,C 0,E1 0.1598,E2 90.0715} C_DIS
LIN {X 1.9218,Y -8.2665,Z 11,A -3.0737,B 0,C 0,E1 0.1598,E2 90.0715} C_DIS
LIN {X 0.8946,Y -8.4434,Z 11,A -3.1189,B 0,C 0,E1 0.1598,E2 90.0715} C_DIS
LIN {X 0.0683,Y -8.4871,Z 11,A -3.151,B 0,C 0,E1 0.1598,E2 90.0714} C_DIS
Enddeposition()
LIN {X 0.0003,Y -4.7568,Z 12,A -2.9802,B 0,C 0,E1 0.1598,E2 90.0604} C_DIS
Startdeposition()
$VEL.CP = VEL_PRINT
LIN {X 0.0003,Y -4.7568,Z 12,A -2.9859,B 0,C 0,E1 0.1598,E2 90.0661} C_DIS
LIN {X 0.8632,Y -4.6726,Z 12,A -2.9555,B 0,C 0,E1 0.1598,E2 90.071} C_DIS
LIN {X 1.6156,Y -4.4663,Z 12,A -2.9197,B 0,C 0,E1 0.1598,E2 90.0716} C_DIS
LIN {X 2.1728,Y -4.2257,Z 12,A -2.8891,B 0,C 0,E1 0.1598,E2 90.0716} C_DIS
LIN {X 2.8338,Y -3.8114,Z 12,A -2.8472,B 0,C 0,E1 0.1598,E2 90.0716} C_DIS
LIN {X 3.2982,Y -3.4206,Z 12,A -2.8136,B 0,C 0,E1 0.1598,E2 90.0717} C_DIS
LIN {X 3.7598,Y -2.9029,Z 12,A -2.7746,B 0,C 0,E1 0.1598,E2 90.0717} C_DIS
LIN {X 4.1427,Y -2.3247,Z 12,A -2.736,B 0,C 0,E1 0.1598,E2 90.0717} C_DIS
LIN {X 4.4369,Y -1.6968,Z 12,A -2.6985,B 0,C 0,E1 0.1598,E2 90.0717} C_DIS
LIN {X 4.6369,Y -1.0327,Z 12,A -2.6629,B 0,C 0,E1 0.1598,E2 90.0717} C_DIS
LIN {X 4.7377,Y -0.3466,Z 12,A -2.6301,B 0,C 0,E1 0.1598,E2 90.0718} C_DIS
LIN {X 4.738,Y 0.3469,Z 12,A -2.6007,B 0,C 0,E1 0.1598,E2 90.0718} C_DIS
LIN {X 4.6365,Y 1.0329,Z 12,A -2.5753,B 0,C 0,E1 0.1598,E2 90.0718} C_DIS
LIN {X 4.4366,Y 1.697,Z 12,A -2.5546,B 0,C 0,E1 0.1598,E2 90.0719} C_DIS
LIN {X 4.1427,Y 2.325,Z 12,A -2.5388,B 0,C 0,E1 0.1598,E2 90.0719} C_DIS
LIN {X 3.7594,Y 2.9029,Z 12,A -2.5285,B 0,C 0,E1 0.1598,E2 90.072} C_DIS
LIN {X 3.2963,Y 3.419,Z 12,A -2.5237,B 0,C 0,E1 0.1598,E2 90.072} C_DIS
LIN {X 2.7649,Y 3.8648,Z 12,A -2.5245,B 0,C 0,E1 0.1598,E2 90.072} C_DIS
LIN {X 2.1719,Y 4.2247,Z 12,A -2.5311,B 0,C 0,E1 0.1598,E2 90.0721} C_DIS
LIN {X 1.5333,Y 4.495,Z 12,A -2.5433,B 0,C 0,E1 0.1598,E2 90.0721} C_DIS
LIN {X 0.8625,Y 4.671,Z 12,A -2.5606,B 0,C 0,E1 0.1598,E2 90.0721} C_DIS
LIN {X 0.1733,Y 4.7492,Z 12,A -2.5827,B 0,C 0,E1 0.1598,E2 90.0721} C_DIS
LIN {X -0.5199,Y 4.7233,Z 12,A -2.6094,B 0,C 0,E1 0.1598,E2 90.0721} C_DIS
LIN {X -1.202,Y 4.5969,Z 12,A -2.6399,B 0,C 0,E1 0.1598,E2 90.0721} C_DIS
LIN {X -1.8586,Y 4.3733,Z 12,A -2.6735,B 0,C 0,E1 0.1598,E2 90.072} C_DIS
LIN {X -2.4744,Y 4.0544,Z 12,A -2.7096,B 0,C 0,E1 0.1598,E2 90.072} C_DIS
LIN {X -3.0385,Y 3.6512,Z 12,A -2.7474,B 0,C 0,E1 0.1598,E2 90.0718} C_DIS
LIN {X -3.5377,Y 3.1698,Z 12,A -2.786,B 0,C 0,E1 0.1598,E2 90.0718} C_DIS
LIN {X -3.9616,Y 2.621,Z 12,A -2.8248,B 0,C 0,E1 0.1598,E2 90.0717} C_DIS
LIN {X -4.3022,Y 2.0167,Z 12,A -2.8628,B 0,C 0,E1 0.1598,E2 90.0716} C_DIS
LIN {X -4.5493,Y 1.3685,Z 12,A -2.8992,B 0,C 0,E1 0.1598,E2 90.0715} C_DIS
LIN {X -4.7006,Y 0.6916,Z 12,A -2.9332,B 0,C 0,E1 0.1598,E2 90.0715} C_DIS
LIN {X -4.7526,Y -0.0001,Z 12,A -2.9643,B 0,C 0,E1 0.1598,E2 90.0714} C_DIS
LIN {X -4.6992,Y -0.6917,Z 12,A -2.9915,B 0,C 0,E1 0.1598,E2 90.0714} C_DIS
LIN {X -4.5485,Y -1.3684,Z 12,A -3.0145,B 0,C 0,E1 0.1598,E2 90.0714} C_DIS
LIN {X -4.3025,Y -2.0171,Z 12,A -3.0329,B 0,C 0,E1 0.1598,E2 90.0714} C_DIS
LIN {X -3.9609,Y -2.6206,Z 12,A -3.0458,B 0,C 0,E1 0.1598,E2 90.0714} C_DIS
LIN {X -3.5369,Y -3.1694,Z 12,A -3.0535,B 0,C 0,E1 0.1598,E2 90.0714} C_DIS
LIN {X -3.0389,Y -3.6523,Z 12,A -3.0556,B 0,C 0,E1 0.1598,E2 90.0714} C_DIS
LIN {X -2.4753,Y -4.0566,Z 12,A -3.052,B 0,C 0,E1 0.1598,E2 90.0714} C_DIS
LIN {X -1.8578,Y -4.3727,Z 12,A -3.0427,B 0,C 0,E1 0.1598,E2 90.0714} C_DIS
LIN {X -1.2013,Y -4.5965,Z 12,A -3.0281,B 0,C 0,E1 0.1598,E2 90.0715} C_DIS
LIN {X -0.5193,Y -4.7224,Z 12,A -3.0084,B 0,C 0,E1 0.1598,E2 90.0715} C_DIS
LIN {X -0.5193,Y -4.7224,Z 12,A -3.0084,B 0,C 0,E1 0.1598,E2 90.0715} C_DIS
Enddeposition()
LIN {X 0.0166,Y -5.6864,Z 12,A -3.0286,B 0,C 0,E1 0.1598,E2 90.0704} C_DIS
Startdeposition()
$VEL.CP = VEL_PRINT
LIN {X -0.9593,Y -5.6009,Z 12,A -3.0618,B 0,C 0,E1 0.1598,E2 90.0714} C_DIS
LIN {X -1.7209,Y -5.4157,Z 12,A -3.082,B 0,C 0,E1 0.1598,E2 90.0714} C_DIS
LIN {X -2.4505,Y -5.1288,Z 12,A -3.0966,B 0,C 0,E1 0.1598,E2 90.0714} C_DIS
LIN {X -3.1338,Y -4.744,Z 12,A -3.1054,B 0,C 0,E1 0.1598,E2 90.0714} C_DIS
LIN {X -3.7547,Y -4.2653,Z 12,A -3.1079,B 0,C 0,E1 0.1598,E2 90.0714} C_DIS
LIN {X -4.3063,Y -3.7084,Z 12,A -3.1046,B 0,C 0,E1 0.1598,E2 90.0713} C_DIS
LIN {X -4.7754,Y -3.0804,Z 12,A -3.0953,B 0,C 0,E1 0.1598,E2 90.0713} C_DIS
LIN {X -5.1543,Y -2.3941,Z 12,A -3.0802,B 0,C 0,E1 0.1598,E2 90.0713} C_DIS
LIN {X -5.4375,Y -1.6629,Z 12,A -3.0597,B 0,C 0,E1 0.1598,E2 90.0713} C_DIS
LIN {X -5.6142,Y -0.8988,Z 12,A -3.034,B 0,C 0,E1 0.1598,E2 90.0713} C_DIS
LIN {X -5.683,Y -0.1176,Z 12,A -3.0036,B 0,C 0,E1 0.1598,E2 90.0713} C_DIS
LIN {X -5.603,Y 0.993,Z 12,A -2.9535,B 0,C 0,E1 0.1598,E2 90.071} C_DIS
LIN {X -5.406,Y 1.7751,Z 12,A -2.9136,B 0,C 0,E1 0.1598,E2 90.0714} C_DIS
LIN {X -4.9402,Y 2.8103,Z 12,A -2.8526,B 0,C 0,E1 0.1598,E2 90.0712} C_DIS
LIN {X -4.5125,Y 3.4552,Z 12,A -2.81,B 0,C 0,E1 0.1598,E2 90.0716} C_DIS
LIN {X -4.0011,Y 4.036,Z 12,A -2.7667,B 0,C 0,E1 0.1598,E2 90.0717} C_DIS
LIN {X -3.2627,Y 4.6608,Z 12,A -2.7131,B 0,C 0,E1 0.1598,E2 90.0717} C_DIS
LIN {X -2.0797,Y 5.296,Z 12,A -2.6427,B 0,C 0,E1 0.1598,E2 90.0719} C_DIS
LIN {X -1.0803,Y 5.5797,Z 12,A -2.594,B 0,C 0,E1 0.1598,E2 90.0721} C_DIS
LIN {X -0.255,Y 5.6774,Z 12,A -2.5595,B 0,C 0,E1 0.1598,E2 90.0721} C_DIS
LIN {X 0.5758,Y 5.6547,Z 12,A -2.5298,B 0,C 0,E1 0.1598,E2 90.0721} C_DIS
LIN {X 1.394,Y 5.5089,Z 12,A -2.5057,B 0,C 0,E1 0.1598,E2 90.0722} C_DIS
LIN {X 2.1825,Y 5.2468,Z 12,A -2.4877,B 0,C 0,E1 0.1598,E2 90.0722} C_DIS
LIN {X 2.9241,Y 4.8717,Z 12,A -2.4762,B 0,C 0,E1 0.1598,E2 90.0722} C_DIS
LIN {X 3.6033,Y 4.3929,Z 12,A -2.4714,B 0,C 0,E1 0.1598,E2 90.0722} C_DIS
LIN {X 4.2059,Y 3.8208,Z 12,A -2.4733,B 0,C 0,E1 0.1598,E2 90.0721} C_DIS
LIN {X 4.7178,Y 3.1663,Z 12,A -2.4821,B 0,C 0,E1 0.1598,E2 90.0721} C_DIS
LIN {X 5.1294,Y 2.4444,Z 12,A -2.4975,B 0,C 0,E1 0.1598,E2 90.0719} C_DIS
LIN {X 5.4321,Y 1.6704,Z 12,A -2.5191,B 0,C 0,E1 0.1598,E2 90.0719} C_DIS
LIN {X 5.6162,Y 0.8601,Z 12,A -2.5467,B 0,C 0,E1 0.1598,E2 90.0719} C_DIS
LIN {X 5.6824,Y 0.0318,Z 12,A -2.5793,B 0,C 0,E1 0.1598,E2 90.0718} C_DIS
LIN {X 5.6267,Y -0.7973,Z 12,A -2.6166,B 0,C 0,E1 0.1598,E2 90.0718} C_DIS
LIN {X 5.45,Y -1.6092,Z 12,A -2.6575,B 0,C 0,E1 0.1598,E2 90.0717} C_DIS
LIN {X 5.1564,Y -2.3867,Z 12,A -2.7014,B 0,C 0,E1 0.1598,E2 90.0717} C_DIS
LIN {X 4.7537,Y -3.1136,Z 12,A -2.747,B 0,C 0,E1 0.1598,E2 90.0717} C_DIS
LIN {X 4.2496,Y -3.7743,Z 12,A -2.7936,B 0,C 0,E1 0.1598,E2 90.0717} C_DIS
LIN {X 3.6544,Y -4.3547,Z 12,A -2.8402,B 0,C 0,E1 0.1598,E2 90.0717} C_DIS
LIN {X 2.9805,Y -4.8417,Z 12,A -2.8856,B 0,C 0,E1 0.1598,E2 90.0717} C_DIS
LIN {X 2.2425,Y -5.2246,Z 12,A -2.929,B 0,C 0,E1 0.1598,E2 90.0717} C_DIS
LIN {X 1.4561,Y -5.4944,Z 12,A -2.9693,B 0,C 0,E1 0.1598,E2 90.0716} C_DIS
LIN {X 0.6391,Y -5.6476,Z 12,A -3.0058,B 0,C 0,E1 0.1598,E2 90.0716} C_DIS
LIN {X 0.0166,Y -5.6864,Z 12,A -3.0303,B 0,C 0,E1 0.1598,E2 90.0716} C_DIS
Enddeposition()
LIN {X 0.0166,Y -5.6864,Z 12,A -3.0303,B 0,C 0,E1 0.1598,E2 90.0716} C_DIS
Startdeposition()
$VEL.CP = VEL_PRINT
LIN {X 0.5916,Y -6.5935,Z 12,A -3.0472,B 0,C 0,E1 0.1598,E2 90.0709} C_DIS
LIN {X 1.3136,Y -6.49,Z 12,A -3.0169,B 0,C 0,E1 0.1598,E2 90.0715} C_DIS
LIN {X 2.0189,Y -6.3041,Z 12,A -2.9832,B 0,C 0,E1 0.1598,E2 90.0715} C_DIS
LIN {X 2.7002,Y -6.0439,Z 12,A -2.9471,B 0,C 0,E1 0.1598,E2 90.0716} C_DIS
LIN {X 3.3484,Y -5.7096,Z 12,A -2.9091,B 0,C 0,E1 0.1598,E2 90.0716} C_DIS
LIN {X 3.956,Y -5.3062,Z 12,A -2.8697,B 0,C 0,E1 0.1598,E2 90.0716} C_DIS
LIN {X 4.5161,Y -4.8391,Z 12,A -2.8293,B 0,C 0,E1 0.1598,E2 90.0716} C_DIS
LIN {X 5.0212,Y -4.3131,Z 12,A -2.7883,B 0,C 0,E1 0.1598,E2 90.0717} C_DIS
LIN {X 5.4671,Y -3.736,Z 12,A -2.7474,B 0,C 0,E1 0.1598,E2 90.0717} C_DIS
LIN {X 5.8434,Y -3.1112,Z 12,A -2.707,B 0,C 0,E1 0.1598,E2 90.0717} C_DIS
LIN {X 6.15,Y -2.4493,Z 12,A -2.6677,B 0,C 0,E1 0.1598,E2 90.0717} C_DIS
LIN {X 6.3816,Y -1.7578,Z 12,A -2.6297,B 0,C 0,E1 0.1598,E2 90.0718} C_DIS
LIN {X 6.5371,Y -1.0453,Z 12,A -2.5938,B 0,C 0,E1 0.1598,E2 90.0718} C_DIS
LIN {X 6.6122,Y -0.3199,Z 12,A -2.5602,B 0,C 0,E1 0.1598,E2 90.0718} C_DIS
LIN {X 6.6063,Y 0.4094,Z 12,A -2.5294,B 0,C 0,E1 0.1598,E2 90.0719} C_DIS
LIN {X 6.5207,Y 1.1336,Z 12,A -2.5018,B 0,C 0,E1 0.1598,E2 90.0719} C_DIS
LIN {X 6.3572,Y 1.8443,Z 12,A -2.4777,B 0,C 0,E1 0.1598,E2 90.0719} C_DIS
LIN {X 6.116,Y 2.5326,Z 12,A -2.4574,B 0,C 0,E1 0.1598,E2 90.072} C_DIS
LIN {X 5.8002,Y 3.19,Z 12,A -2.4412,B 0,C 0,E1 0.1598,E2 90.072} C_DIS
LIN {X 5.4127,Y 3.8079,Z 12,A -2.4293,B 0,C 0,E1 0.1598,E2 90.0721} C_DIS
LIN {X 4.9608,Y 4.3802,Z 12,A -2.4218,B 0,C 0,E1 0.1598,E2 90.0721} C_DIS
LIN {X 4.4496,Y 4.9001,Z 12,A -2.4186,B 0,C 0,E1 0.1598,E2 90.0721} C_DIS
LIN {X 3.8838,Y 5.3603,Z 12,A -2.42,B 0,C 0,E1 0.1598,E2 90.0722} C_DIS
LIN {X 3.2704,Y 5.755,Z 12,A -2.426,B 0,C 0,E1 0.1598,E2 90.0722} C_DIS
LIN {X 2.6171,Y 6.0792,Z 12,A -2.4364,B 0,C 0,E1 0.1598,E2 90.0722} C_DIS
LIN {X 1.9328,Y 6.3314,Z 12,A -2.451,B 0,C 0,E1 0.1598,E2 90.0722} C_DIS
LIN {X 1.2243,Y 6.5045,Z 12,A -2.4699,B 0,C 0,E1 0.1598,E2 90.0722} C_DIS
LIN {X 0.5013,Y 6.5988,Z 12,A -2.4926,B 0,C 0,E1 0.1598,E2 90.0722} C_DIS
LIN {X -0.2278,Y 6.6166,Z 12,A -2.5187,B 0,C 0,E1 0.1598,E2 90.0722} C_DIS
LIN {X -0.9543,Y 6.5509,Z 12,A -2.5483,B 0,C 0,E1 0.1598,E2 90.0722} C_DIS
LIN {X -1.6694,Y 6.4081,Z 12,A -2.5807,B 0,C 0,E1 0.1598,E2 90.0722} C_DIS
LIN {X -2.3637,Y 6.1846,Z 12,A -2.6157,B 0,C 0,E1 0.1598,E2 90.0721} C_DIS
LIN {X -3.0287,Y 5.8855,Z 12,A -2.6529,B 0,C 0,E1 0.1598,E2 90.072} C_DIS
LIN {X -3.6576,Y 5.5162,Z 12,A -2.6916,B 0,C 0,E1 0.1598,E2 90.072} C_DIS
LIN {X -4.2432,Y 5.0813,Z 12,A -2.7315,B 0,C 0,E1 0.1598,E2 90.0718} C_DIS
LIN {X -4.776,Y 4.5833,Z 12,A -2.7721,B 0,C 0,E1 0.1598,E2 90.0718} C_DIS
LIN {X -5.2498,Y 4.0288,Z 12,A -2.8129,B 0,C 0,E1 0.1598,E2 90.0717} C_DIS
LIN {X -5.6626,Y 3.4277,Z 12,A -2.8534,B 0,C 0,E1 0.1598,E2 90.0716} C_DIS
LIN {X -6.0065,Y 2.7847,Z 12,A -2.8931,B 0,C 0,E1 0.1598,E2 90.0716} C_DIS
LIN {X -6.2749,Y 2.1066,Z 12,A -2.9315,B 0,C 0,E1 0.1598,E2 90.0714} C_DIS
LIN {X -6.469,Y 1.4037,Z 12,A -2.9683,B 0,C 0,E1 0.1598,E2 90.0714} C_DIS
LIN {X -6.5848,Y 0.6837,Z 12,A -3.0028,B 0,C 0,E1 0.1598,E2 90.0714} C_DIS
LIN {X -6.62,Y -0.0449,Z 12,A -3.0348,B 0,C 0,E1 0.1598,E2 90.0713} C_DIS
LIN {X -6.5739,Y -0.7727,Z 12,A -3.0638,B 0,C 0,E1 0.1598,E2 90.0713} C_DIS
LIN {X -6.4485,Y -1.4912,Z 12,A -3.0895,B 0,C 0,E1 0.1598,E2 90.0712} C_DIS
LIN {X -6.2449,Y -2.1913,Z 12,A -3.1115,B 0,C 0,E1 0.1598,E2 90.0712} C_DIS
LIN {X -5.9656,Y -2.8649,Z 12,A -3.1297,B 0,C 0,E1 0.1598,E2 90.0712} C_DIS
LIN {X -5.6169,Y -3.5055,Z 12,A -3.1439,B 0,C 0,E1 0.1598,E2 90.0712} C_DIS
LIN {X -5.1965,Y -4.1016,Z 12,A -3.1536,B 0,C 0,E1 0.1598,E2 90.0712} C_DIS
LIN {X -4.7135,Y -4.6482,Z 12,A -3.159,B 0,C 0,E1 0.1598,E2 90.0712} C_DIS
LIN {X -4.1733,Y -5.1382,Z 12,A -3.1599,B 0,C 0,E1 0.1598,E2 90.0712} C_DIS
LIN {X -3.5821,Y -5.5652,Z 12,A -3.1563,B 0,C 0,E1 0.1598,E2 90.0712} C_DIS
LIN {X -2.948,Y -5.9253,Z 12,A -3.1482,B 0,C 0,E1 0.1598,E2 90.0713} C_DIS
LIN {X -2.2789,Y -6.2156,Z 12,A -3.136,B 0,C 0,E1 0.1598,E2 90.0713} C_DIS
LIN {X -1.5807,Y -6.4265,Z 12,A -3.1193,B 0,C 0,E1 0.1598,E2 90.0713} C_DIS
LIN {X -0.8643,Y -6.562,Z 12,A -3.0988,B 0,C 0,E1 0.1598,E2 90.0714} C_DIS
LIN {X 0.0452,Y -6.6236,Z 12,A -3.0681,B 0,C 0,E1 0.1598,E2 90.0714} C_DIS
Enddeposition()
LIN {X 0.0452,Y -6.6236,Z 12,A -3.0681,B 0,C 0,E1 0.1598,E2 90.0714} C_DIS
Startdeposition()
$VEL.CP = VEL_PRINT
LIN {X -0.4653,Y -7.5396,Z 12,A -3.1252,B 0,C 0,E1 0.1598,E2 90.0709} C_DIS
LIN {X -1.1819,Y -7.4588,Z 12,A -3.1486,B 0,C 0,E1 0.1598,E2 90.0713} C_DIS
LIN {X -2.0637,Y -7.2713,Z 12,A -3.173,B 0,C 0,E1 0.1598,E2 90.0713} C_DIS
LIN {X -3.1047,Y -6.8856,Z 12,A -3.1948,B 0,C 0,E1 0.1598,E2 90.0713} C_DIS
LIN {X -3.8159,Y -6.5184,Z 12,A -3.2053,B 0,C 0,E1 0.1598,E2 90.0713} C_DIS
LIN {X -4.4845,Y -6.0782,Z 12,A -3.2112,B 0,C 0,E1 0.1598,E2 90.0712} C_DIS
LIN {X -5.1025,Y -5.5693,Z 12,A -3.2124,B 0,C 0,E1 0.1598,E2 90.0712} C_DIS
LIN {X -5.871,Y -4.7589,Z 12,A -3.2062,B 0,C 0,E1 0.1598,E2 90.071} C_DIS
LIN {X -6.4677,Y -3.8989,Z 12,A -3.1918,B 0,C 0,E1 0.1598,E2 90.071} C_DIS
LIN {X -6.9949,Y -2.8608,Z 12,A -3.1672,B 0,C 0,E1 0.1598,E2 90.0708} C_DIS
LIN {X -7.3368,Y -1.7962,Z 12,A -3.1349,B 0,C 0,E1 0.1598,E2 90.0708} C_DIS
LIN {X -7.5341,Y -0.5922,Z 12,A -3.0913,B 0,C 0,E1 0.1598,E2 90.0708} C_DIS
LIN {X -7.5416,Y 0.4173,Z 12,A -3.0492,B 0,C 0,E1 0.1598,E2 90.071} C_DIS
LIN {X -7.4524,Y 1.2198,Z 12,A -3.0123,B 0,C 0,E1 0.1598,E2 90.0712} C_DIS
LIN {X -7.2794,Y 2.0085,Z 12,A -2.9728,B 0,C 0,E1 0.1598,E2 90.0712} C_DIS
LIN {X -7.025,Y 2.7748,Z 12,A -2.9311,B 0,C 0,E1 0.1598,E2 90.0714} C_DIS
LIN {X -6.549,Y 3.7728,Z 12,A -2.8714,B 0,C 0,E1 0.1598,E2 90.0713} C_DIS
LIN {X -6.0376,Y 4.5385,Z 12,A -2.8205,B 0,C 0,E1 0.1598,E2 90.0715} C_DIS
LIN {X -5.5669,Y 5.1052,Z 12,A -2.7794,B 0,C 0,E1 0.1598,E2 90.0717} C_DIS
LIN {X -5.0429,Y 5.623,Z 12,A -2.7383,B 0,C 0,E1 0.1598,E2 90.0717} C_DIS
LIN {X -4.4717,Y 6.0882,Z 12,A -2.6977,B 0,C 0,E1 0.1598,E2 90.0719} C_DIS
LIN {X -3.5539,Y 6.6693,Z 12,A -2.6393,B 0,C 0,E1 0.1598,E2 90.0719} C_DIS
LIN {X -2.4675,Y 7.1396,Z 12,A -2.5794,B 0,C 0,E1 0.1598,E2 90.072} C_DIS
LIN {X -1.7791,Y 7.3454,Z 12,A -2.5454,B 0,C 0,E1 0.1598,E2 90.0721} C_DIS
LIN {X -0.7724,Y 7.5177,Z 12,A -2.501,B 0,C 0,E1 0.1598,E2 90.0722} C_DIS
LIN {X 0.2418,Y 7.5534,Z 12,A -2.462,B 0,C 0,E1 0.1598,E2 90.0722} C_DIS
LIN {X 1.4549,Y 7.4121,Z 12,A -2.4232,B 0,C 0,E1 0.1598,E2 90.0723} C_DIS
LIN {X 2.189,Y 7.233,Z 12,A -2.4037,B 0,C 0,E1 0.1598,E2 90.0723} C_DIS
LIN {X 3.0933,Y 6.89,Z 12,A -2.3847,B 0,C 0,E1 0.1598,E2 90.0723} C_DIS
LIN {X 3.7822,Y 6.5381,Z 12,A -2.3742,B 0,C 0,E1 0.1598,E2 90.0723} C_DIS
LIN {X 4.4312,Y 6.1168,Z 12,A -2.368,B 0,C 0,E1 0.1598,E2 90.0723} C_DIS
LIN {X 5.0334,Y 5.6309,Z 12,A -2.3664,B 0,C 0,E1 0.1598,E2 90.0723} C_DIS
LIN {X 5.5829,Y 5.0862,Z 12,A -2.3691,B 0,C 0,E1 0.1598,E2 90.0723} C_DIS
LIN {X 6.0739,Y 4.4883,Z 12,A -2.3763,B 0,C 0,E1 0.1598,E2 90.0722} C_DIS
LIN {X 6.5019,Y 3.8438,Z 12,A -2.3878,B 0,C 0,E1 0.1598,E2 90.0722} C_DIS
LIN {X 6.8614,Y 3.1585,Z 12,A -2.4036,B 0,C 0,E1 0.1598,E2 90.0721} C_DIS
LIN {X 7.2484,Y 2.1398,Z 12,A -2.4323,B 0,C 0,E1 0.1598,E2 90.0718} C_DIS
LIN {X 7.4648,Y 1.1755,Z 12,A -2.4653,B 0,C 0,E1 0.1598,E2 90.0718} C_DIS
LIN {X 7.5568,Y 0.0746,Z 12,A -2.5085,B 0,C 0,E1 0.1598,E2 90.0715} C_DIS
LIN {X 7.5145,Y -0.8007,Z 12,A -2.5474,B 0,C 0,E1 0.1598,E2 90.0716} C_DIS
LIN {X 7.2743,Y -2.0513,Z 12,A -2.609,B 0,C 0,E1 0.1598,E2 90.0713} C_DIS
LIN {X 6.8658,Y -3.16,Z 12,A -2.6713,B 0,C 0,E1 0.1598,E2 90.0713} C_DIS
LIN {X 6.2658,Y -4.2246,Z 12,A -2.7387,B 0,C 0,E1 0.1598,E2 90.0713} C_DIS
LIN {X 5.0158,Y -5.6533,Z 12,A -2.8448,B 0,C 0,E1 0.1598,E2 90.0709} C_DIS
LIN {X 3.9917,Y -6.4161,Z 12,A -2.9154,B 0,C 0,E1 0.1598,E2 90.0714} C_DIS
LIN {X 3.1605,Y -6.8656,Z 12,A -2.9652,B 0,C 0,E1 0.1598,E2 90.0715} C_DIS
LIN {X 2.0724,Y -7.2631,Z 12,A -3.022,B 0,C 0,E1 0.1598,E2 90.0715} C_DIS
LIN {X 0.9085,Y -7.5022,Z 12,A -3.0749,B 0,C 0,E1 0.1598,E2 90.0715} C_DIS
LIN {X 0.0754,Y -7.5549,Z 12,A -3.1076,B 0,C 0,E1 0.1598,E2 90.0715} C_DIS
Enddeposition()
LIN {X 0.0754,Y -7.5549,Z 12,A -3.1076,B 0,C 0,E1 0.1598,E2 90.0715} C_DIS
Startdeposition()
$VEL.CP = VEL_PRINT
LIN {X 0.7304,Y -8.4559,Z 12,A -3.1215,B 0,C 0,E1 0.1598,E2 90.0709} C_DIS
LIN {X 1.5534,Y -8.3431,Z 12,A -3.087,B 0,C 0,E1 0.1598,E2 90.0714} C_DIS
LIN {X 2.3616,Y -8.151,Z 12,A -3.0493,B 0,C 0,E1 0.1598,E2 90.0714} C_DIS
LIN {X 3.1472,Y -7.8811,Z 12,A -3.009,B 0,C 0,E1 0.1598,E2 90.0715} C_DIS
LIN {X 3.9028,Y -7.5358,Z 12,A -2.9666,B 0,C 0,E1 0.1598,E2 90.0715} C_DIS
LIN {X 4.621,Y -7.1184,Z 12,A -2.9225,B 0,C 0,E1 0.1598,E2 90.0715} C_DIS
LIN {X 5.2951,Y -6.6329,Z 12,A -2.8772,B 0,C 0,E1 0.1598,E2 90.0716} C_DIS
LIN {X 5.9188,Y -6.0841,Z 12,A -2.8309,B 0,C 0,E1 0.1598,E2 90.0716} C_DIS
LIN {X 6.4859,Y -5.4769,Z 12,A -2.7843,B 0,C 0,E1 0.1598,E2 90.0716} C_DIS
LIN {X 6.9907,Y -4.817,Z 12,A -2.7377,B 0,C 0,E1 0.1598,E2 90.0716} C_DIS
LIN {X 7.428,Y -4.1106,Z 12,A -2.6915,B 0,C 0,E1 0.1598,E2 90.0717} C_DIS
LIN {X 7.8762,Y -3.1738,Z 12,A -2.635,B 0,C 0,E1 0.1598,E2 90.0715} C_DIS
LIN {X 8.2376,Y -2.0443,Z 12,A -2.5735,B 0,C 0,E1 0.1598,E2 90.0715} C_DIS
LIN {X 8.4025,Y -1.1931,Z 12,A -2.5315,B 0,C 0,E1 0.1598,E2 90.0718} C_DIS
LIN {X 8.4921,Y -0.0195,Z 12,A -2.4781,B 0,C 0,E1 0.1598,E2 90.0716} C_DIS
LIN {X 8.4113,Y 1.1287,Z 12,A -2.4322,B 0,C 0,E1 0.1598,E2 90.0716} C_DIS
LIN {X 8.2599,Y 1.9481,Z 12,A -2.4033,B 0,C 0,E1 0.1598,E2 90.072} C_DIS
LIN {X 8.029,Y 2.7487,Z 12,A -2.3779,B 0,C 0,E1 0.1598,E2 90.072} C_DIS
LIN {X 7.7208,Y 3.5228,Z 12,A -2.3564,B 0,C 0,E1 0.1598,E2 90.072} C_DIS
LIN {X 7.3382,Y 4.2631,Z 12,A -2.3391,B 0,C 0,E1 0.1598,E2 90.0721} C_DIS
LIN {X 6.8851,Y 4.9624,Z 12,A -2.3262,B 0,C 0,E1 0.1598,E2 90.0721} C_DIS
LIN {X 6.3657,Y 5.614,Z 12,A -2.3177,B 0,C 0,E1 0.1598,E2 90.0722} C_DIS
LIN {X 5.7851,Y 6.2117,Z 12,A -2.3139,B 0,C 0,E1 0.1598,E2 90.0722} C_DIS
LIN {X 5.1484,Y 6.7492,Z 12,A -2.3146,B 0,C 0,E1 0.1598,E2 90.0723} C_DIS
LIN {X 4.4619,Y 7.2217,Z 12,A -2.32,B 0,C 0,E1 0.1598,E2 90.0723} C_DIS
LIN {X 3.7322,Y 7.6242,Z 12,A -2.3299,B 0,C 0,E1 0.1598,E2 90.0723} C_DIS
LIN {X 2.9667,Y 7.9534,Z 12,A -2.3443,B 0,C 0,E1 0.1598,E2 90.0723} C_DIS
LIN {X 2.1726,Y 8.2063,Z 12,A -2.363,B 0,C 0,E1 0.1598,E2 90.0723} C_DIS
LIN {X 1.3576,Y 8.3802,Z 12,A -2.3858,B 0,C 0,E1 0.1598,E2 90.0723} C_DIS
LIN {X 0.5294,Y 8.4725,Z 12,A -2.4125,B 0,C 0,E1 0.1598,E2 90.0723} C_DIS
LIN {X -0.3038,Y 8.4822,Z 12,A -2.4428,B 0,C 0,E1 0.1598,E2 90.0723} C_DIS
LIN {X -1.134,Y 8.4107,Z 12,A -2.4765,B 0,C 0,E1 0.1598,E2 90.0723} C_DIS
LIN {X -1.9532,Y 8.2587,Z 12,A -2.5132,B 0,C 0,E1 0.1598,E2 90.0723} C_DIS
LIN {X -2.7537,Y 8.0273,Z 12,A -2.5525,B 0,C 0,E1 0.1598,E2 90.0721} C_DIS
LIN {X -3.5277,Y 7.7186,Z 12,A -2.594,B 0,C 0,E1 0.1598,E2 90.0721} C_DIS
LIN {X -4.2677,Y 7.3355,Z 12,A -2.6375,B 0,C 0,E1 0.1598,E2 90.072} C_DIS
LIN {X -4.9667,Y 6.8819,Z 12,A -2.6823,B 0,C 0,E1 0.1598,E2 90.0719} C_DIS
LIN {X -5.618,Y 6.3621,Z 12,A -2.7282,B 0,C 0,E1 0.1598,E2 90.0719} C_DIS
LIN {X -6.2153,Y 5.7811,Z 12,A -2.7747,B 0,C 0,E1 0.1598,E2 90.0717} C_DIS
LIN {X -6.7525,Y 5.1441,Z 12,A -2.8212,B 0,C 0,E1 0.1598,E2 90.0717} C_DIS
LIN {X -7.2246,Y 4.4574,Z 12,A -2.8675,B 0,C 0,E1 0.1598,E2 90.0715} C_DIS
LIN {X -7.6261,Y 3.7272,Z 12,A -2.913,B 0,C 0,E1 0.1598,E2 90.0715} C_DIS
LIN {X -7.9548,Y 2.9615,Z 12,A -2.9573,B 0,C 0,E1 0.1598,E2 90.0713} C_DIS
LIN {X -8.2075,Y 2.1674,Z 12,A -3,B 0,C 0,E1 0.1598,E2 90.0713} C_DIS
LIN {X -8.3811,Y 1.3523,Z 12,A -3.0406,B 0,C 0,E1 0.1598,E2 90.0712} C_DIS
LIN {X -8.4879,Y 0.2129,Z 12,A -3.0922,B 0,C 0,E1 0.1598,E2 90.0708} C_DIS
LIN {X -8.4599,Y -0.7393,Z 12,A -3.1314,B 0,C 0,E1 0.1598,E2 90.0709} C_DIS
LIN {X -8.2769,Y -1.8773,Z 12,A -3.1724,B 0,C 0,E1 0.1598,E2 90.0706} C_DIS
LIN {X -8.0519,Y -2.685,Z 12,A -3.1984,B 0,C 0,E1 0.1598,E2 90.071} C_DIS
LIN {X -7.7476,Y -3.4663,Z 12,A -3.2202,B 0,C 0,E1 0.1598,E2 90.071} C_DIS
LIN {X -7.3679,Y -4.2139,Z 12,A -3.2378,B 0,C 0,E1 0.1598,E2 90.071} C_DIS
LIN {X -6.916,Y -4.9202,Z 12,A -3.251,B 0,C 0,E1 0.1598,E2 90.071} C_DIS
LIN {X -6.3958,Y -5.5778,Z 12,A -3.2597,B 0,C 0,E1 0.1598,E2 90.071} C_DIS
LIN {X -5.8154,Y -6.1828,Z 12,A -3.264,B 0,C 0,E1 0.1598,E2 90.071} C_DIS
LIN {X -5.1781,Y -6.7276,Z 12,A -3.2636,B 0,C 0,E1 0.1598,E2 90.071} C_DIS
LIN {X -4.4891,Y -7.2054,Z 12,A -3.2586,B 0,C 0,E1 0.1598,E2 90.0711} C_DIS
LIN {X -3.4239,Y -7.7699,Z 12,A -3.2434,B 0,C 0,E1 0.1598,E2 90.0711} C_DIS
LIN {X -2.4472,Y -8.1264,Z 12,A -3.2227,B 0,C 0,E1 0.1598,E2 90.0712} C_DIS
LIN {X -1.6402,Y -8.3277,Z 12,A -3.2017,B 0,C 0,E1 0.1598,E2 90.0712} C_DIS
LIN {X -0.6099,Y -8.4687,Z 12,A -3.1699,B 0,C 0,E1 0.1598,E2 90.0713} C_DIS
LIN {X 0.108,Y -8.4884,Z 12,A -3.1445,B 0,C 0,E1 0.1598,E2 90.0713} C_DIS
Enddeposition()
LIN {X 0.0003,Y -4.7572,Z 13,A -2.9751,B 0,C 0,E1 0.1598,E2 90.0603} C_DIS
Startdeposition()
$VEL.CP = VEL_PRINT
LIN {X 0.0003,Y -4.7572,Z 13,A -2.9807,B 0,C 0,E1 0.1598,E2 90.0661} C_DIS
LIN {X -0.8628,Y -4.6738,Z 13,A -3.0138,B 0,C 0,E1 0.1598,E2 90.0709} C_DIS
LIN {X -1.5339,Y -4.4975,Z 13,A -3.0315,B 0,C 0,E1 0.1598,E2 90.0715} C_DIS
LIN {X -2.1719,Y -4.2256,Z 13,A -3.0435,B 0,C 0,E1 0.1598,E2 90.0715} C_DIS
LIN {X -2.764,Y -3.8644,Z 13,A -3.0499,B 0,C 0,E1 0.1598,E2 90.0715} C_DIS
LIN {X -3.2977,Y -3.4211,Z 13,A -3.0507,B 0,C 0,E1 0.1598,E2 90.0714} C_DIS
LIN {X -3.7595,Y -2.9035,Z 13,A -3.0458,B 0,C 0,E1 0.1598,E2 90.0714} C_DIS
LIN {X -4.1834,Y -2.2486,Z 13,A -3.0336,B 0,C 0,E1 0.1598,E2 90.0713} C_DIS
LIN {X -4.4368,Y -1.6972,Z 13,A -3.0197,B 0,C 0,E1 0.1598,E2 90.0713} C_DIS
LIN {X -4.6368,Y -1.0332,Z 13,A -2.999,B 0,C 0,E1 0.1598,E2 90.0713} C_DIS
LIN {X -4.7377,Y -0.3471,Z 13,A -2.9738,B 0,C 0,E1 0.1598,E2 90.0713} C_DIS
LIN {X -4.7381,Y 0.3464,Z 13,A -2.9445,B 0,C 0,E1 0.1598,E2 90.0713} C_DIS
LIN {X -4.6366,Y 1.0324,Z 13,A -2.9118,B 0,C 0,E1 0.1598,E2 90.0714} C_DIS
LIN {X -4.4369,Y 1.6965,Z 13,A -2.8765,B 0,C 0,E1 0.1598,E2 90.0715} C_DIS
LIN {X -4.143,Y 2.3246,Z 13,A -2.8392,B 0,C 0,E1 0.1598,E2 90.0715} C_DIS
LIN {X -3.7616,Y 2.9039,Z 13,A -2.8008,B 0,C 0,E1 0.1598,E2 90.0717} C_DIS
LIN {X -3.2986,Y 3.4205,Z 13,A -2.7619,B 0,C 0,E1 0.1598,E2 90.0717} C_DIS
LIN {X -2.7653,Y 3.8645,Z 13,A -2.7236,B 0,C 0,E1 0.1598,E2 90.0718} C_DIS
LIN {X -2.173,Y 4.2253,Z 13,A -2.6866,B 0,C 0,E1 0.1598,E2 90.0719} C_DIS
LIN {X -1.534,Y 4.4953,Z 13,A -2.6516,B 0,C 0,E1 0.1598,E2 90.072} C_DIS
LIN {X -0.863,Y 4.6706,Z 13,A -2.6195,B 0,C 0,E1 0.1598,E2 90.072} C_DIS
LIN {X -0.1739,Y 4.7489,Z 13,A -2.5908,B 0,C 0,E1 0.1598,E2 90.0721} C_DIS
LIN {X 0.5194,Y 4.7234,Z 13,A -2.5663,B 0,C 0,E1 0.1598,E2 90.0721} C_DIS
LIN {X 1.2015,Y 4.5972,Z 13,A -2.5465,B 0,C 0,E1 0.1598,E2 90.0721} C_DIS
LIN {X 1.8579,Y 4.3731,Z 13,A -2.5318,B 0,C 0,E1 0.1598,E2 90.0721} C_DIS
LIN {X 2.4746,Y 4.0555,Z 13,A -2.5224,B 0,C 0,E1 0.1598,E2 90.0721} C_DIS
LIN {X 3.169,Y 3.5372,Z 13,A -2.5187,B 0,C 0,E1 0.1598,E2 90.0721} C_DIS
LIN {X 3.6503,Y 3.0381,Z 13,A -2.5221,B 0,C 0,E1 0.1598,E2 90.0721} C_DIS
LIN {X 4.0539,Y 2.4744,Z 13,A -2.5311,B 0,C 0,E1 0.1598,E2 90.0721} C_DIS
LIN {X 4.4381,Y 1.6976,Z 13,A -2.5497,B 0,C 0,E1 0.1598,E2 90.0719} C_DIS
LIN {X 4.6541,Y 0.9481,Z 13,A -2.5735,B 0,C 0,E1 0.1598,E2 90.0718} C_DIS
LIN {X 4.7377,Y 0.347,Z 13,A -2.596,B 0,C 0,E1 0.1598,E2 90.0718} C_DIS
LIN {X 4.7377,Y -0.3465,Z 13,A -2.6254,B 0,C 0,E1 0.1598,E2 90.0718} C_DIS
LIN {X 4.6367,Y -1.0326,Z 13,A -2.6582,B 0,C 0,E1 0.1598,E2 90.0718} C_DIS
LIN {X 4.4368,Y -1.6966,Z 13,A -2.6937,B 0,C 0,E1 0.1598,E2 90.0718} C_DIS
LIN {X 4.1425,Y -2.3245,Z 13,A -2.7312,B 0,C 0,E1 0.1598,E2 90.0718} C_DIS
LIN {X 3.7616,Y -2.9041,Z 13,A -2.7698,B 0,C 0,E1 0.1598,E2 90.0718} C_DIS
LIN {X 3.2982,Y -3.4204,Z 13,A -2.8088,B 0,C 0,E1 0.1598,E2 90.0717} C_DIS
LIN {X 2.7649,Y -3.864,Z 13,A -2.8472,B 0,C 0,E1 0.1598,E2 90.0717} C_DIS
LIN {X 2.1718,Y -4.2236,Z 13,A -2.8843,B 0,C 0,E1 0.1598,E2 90.0717} C_DIS
LIN {X 1.5337,Y -4.4947,Z 13,A -2.9192,B 0,C 0,E1 0.1598,E2 90.0717} C_DIS
LIN {X 0.8633,Y -4.6722,Z 13,A -2.9514,B 0,C 0,E1 0.1598,E2 90.0717} C_DIS
LIN {X 0.0003,Y -4.7572,Z 13,A -2.9867,B 0,C 0,E1 0.1598,E2 90.0716} C_DIS
Enddeposition()
LIN {X 0.0003,Y -4.7572,Z 13,A -2.9867,B 0,C 0,E1 0.1598,E2 90.0716} C_DIS
Startdeposition()
$VEL.CP = VEL_PRINT
LIN {X 0.5681,Y -5.6548,Z 13,A -3.0034,B 0,C 0,E1 0.1598,E2 90.071} C_DIS
LIN {X 1.3183,Y -5.5308,Z 13,A -2.9712,B 0,C 0,E1 0.1598,E2 90.0716} C_DIS
LIN {X 2.044,Y -5.3036,Z 13,A -2.9349,B 0,C 0,E1 0.1598,E2 90.0716} C_DIS
LIN {X 2.7327,Y -4.9822,Z 13,A -2.896,B 0,C 0,E1 0.1598,E2 90.0716} C_DIS
LIN {X 3.3743,Y -4.5744,Z 13,A -2.8551,B 0,C 0,E1 0.1598,E2 90.0716} C_DIS
LIN {X 3.9543,Y -4.0828,Z 13,A -2.8129,B 0,C 0,E1 0.1598,E2 90.0717} C_DIS
LIN {X 4.4643,Y -3.519,Z 13,A -2.7702,B 0,C 0,E1 0.1598,E2 90.0717} C_DIS
LIN {X 4.8945,Y -2.892,Z 13,A -2.7277,B 0,C 0,E1 0.1598,E2 90.0717} C_DIS
LIN {X 5.2368,Y -2.2131,Z 13,A -2.6863,B 0,C 0,E1 0.1598,E2 90.0717} C_DIS
LIN {X 5.4831,Y -1.4938,Z 13,A -2.6467,B 0,C 0,E1 0.1598,E2 90.0717} C_DIS
LIN {X 5.6357,Y -0.749,Z 13,A -2.6094,B 0,C 0,E1 0.1598,E2 90.0717} C_DIS
LIN {X 5.6865,Y 0.0098,Z 13,A -2.5753,B 0,C 0,E1 0.1598,E2 90.0718} C_DIS
LIN {X 5.6087,Y 0.9572,Z 13,A -2.5377,B 0,C 0,E1 0.1598,E2 90.0716} C_DIS
LIN {X 5.1954,Y 2.3211,Z 13,A -2.4946,B 0,C 0,E1 0.1598,E2 90.0711} C_DIS
LIN {X 4.8945,Y 2.8902,Z 13,A -2.4823,B 0,C 0,E1 0.1598,E2 90.072} C_DIS
LIN {X 4.4046,Y 3.5941,Z 13,A -2.4706,B 0,C 0,E1 0.1598,E2 90.072} C_DIS
LIN {X 3.8132,Y 4.2147,Z 13,A -2.4661,B 0,C 0,E1 0.1598,E2 90.072} C_DIS
LIN {X 3.1364,Y 4.7412,Z 13,A -2.4689,B 0,C 0,E1 0.1598,E2 90.0721} C_DIS
LIN {X 2.3878,Y 5.1594,Z 13,A -2.4788,B 0,C 0,E1 0.1598,E2 90.0721} C_DIS
LIN {X 1.5846,Y 5.4599,Z 13,A -2.4958,B 0,C 0,E1 0.1598,E2 90.0721} C_DIS
LIN {X 0.7453,Y 5.6366,Z 13,A -2.5193,B 0,C 0,E1 0.1598,E2 90.0721} C_DIS
LIN {X -0.1109,Y 5.6836,Z 13,A -2.5489,B 0,C 0,E1 0.1598,E2 90.0721} C_DIS
LIN {X -0.9646,Y 5.6023,Z 13,A -2.5839,B 0,C 0,E1 0.1598,E2 90.0721} C_DIS
LIN {X -1.7961,Y 5.3928,Z 13,A -2.6234,B 0,C 0,E1 0.1598,E2 90.0721} C_DIS
LIN {X -2.5863,Y 5.0603,Z 13,A -2.6665,B 0,C 0,E1 0.1598,E2 90.072} C_DIS
LIN {X -3.3181,Y 4.6138,Z 13,A -2.7123,B 0,C 0,E1 0.1598,E2 90.0719} C_DIS
LIN {X -3.976,Y 4.0642,Z 13,A -2.7596,B 0,C 0,E1 0.1598,E2 90.0717} C_DIS
LIN {X -4.4855,Y 3.4998,Z 13,A -2.8021,B 0,C 0,E1 0.1598,E2 90.0716} C_DIS
LIN {X -5.0017,Y 2.6983,Z 13,A -2.8549,B 0,C 0,E1 0.1598,E2 90.0715} C_DIS
LIN {X -5.3188,Y 2.0047,Z 13,A -2.8958,B 0,C 0,E1 0.1598,E2 90.0715} C_DIS
LIN {X -5.5407,Y 1.2748,Z 13,A -2.9347,B 0,C 0,E1 0.1598,E2 90.0714} C_DIS
LIN {X -5.661,Y 0.5214,Z 13,A -2.9709,B 0,C 0,E1 0.1598,E2 90.0714} C_DIS
LIN {X -5.6777,Y -0.241,Z 13,A -3.0036,B 0,C 0,E1 0.1598,E2 90.0713} C_DIS
LIN {X -5.5368,Y -1.3148,Z 13,A -3.0435,B 0,C 0,E1 0.1598,E2 90.071} C_DIS
LIN {X -5.2219,Y -2.2453,Z 13,A -3.0713,B 0,C 0,E1 0.1598,E2 90.071} C_DIS
LIN {X -4.8618,Y -2.9436,Z 13,A -3.0877,B 0,C 0,E1 0.1598,E2 90.0712} C_DIS
LIN {X -4.4104,Y -3.5867,Z 13,A -3.0983,B 0,C 0,E1 0.1598,E2 90.0712} C_DIS
LIN {X -3.8749,Y -4.162,Z 13,A -3.103,B 0,C 0,E1 0.1598,E2 90.0712} C_DIS
LIN {X -2.9461,Y -4.8673,Z 13,A -3.0986,B 0,C 0,E1 0.1598,E2 90.0712} C_DIS
LIN {X -2.0388,Y -5.3119,Z 13,A -3.0842,B 0,C 0,E1 0.1598,E2 90.0714} C_DIS
LIN {X -1.0613,Y -5.5907,Z 13,A -3.0602,B 0,C 0,E1 0.1598,E2 90.0714} C_DIS
LIN {X -0.0014,Y -5.6857,Z 13,A -3.0254,B 0,C 0,E1 0.1598,E2 90.0715} C_DIS
Enddeposition()
LIN {X -0.0014,Y -5.6857,Z 13,A -3.0254,B 0,C 0,E1 0.1598,E2 90.0715} C_DIS
Startdeposition()
$VEL.CP = VEL_PRINT
LIN {X -0.5204,Y -6.5979,Z 13,A -3.0826,B 0,C 0,E1 0.1598,E2 90.0709} C_DIS
LIN {X -1.2288,Y -6.5053,Z 13,A -3.1052,B 0,C 0,E1 0.1598,E2 90.0714} C_DIS
LIN {X -1.9228,Y -6.3354,Z 13,A -3.1235,B 0,C 0,E1 0.1598,E2 90.0714} C_DIS
LIN {X -2.594,Y -6.0901,Z 13,A -3.1377,B 0,C 0,E1 0.1598,E2 90.0714} C_DIS
LIN {X -3.235,Y -5.7746,Z 13,A -3.1479,B 0,C 0,E1 0.1598,E2 90.0714} C_DIS
LIN {X -3.8388,Y -5.3928,Z 13,A -3.1539,B 0,C 0,E1 0.1598,E2 90.0713} C_DIS
LIN {X -4.3972,Y -4.9472,Z 13,A -3.1555,B 0,C 0,E1 0.1598,E2 90.0713} C_DIS
LIN {X -4.9052,Y -4.4448,Z 13,A -3.1529,B 0,C 0,E1 0.1598,E2 90.0713} C_DIS
LIN {X -5.3557,Y -3.8902,Z 13,A -3.146,B 0,C 0,E1 0.1598,E2 90.0713} C_DIS
LIN {X -5.7427,Y -3.2898,Z 13,A -3.1349,B 0,C 0,E1 0.1598,E2 90.0713} C_DIS
LIN {X -6.0641,Y -2.6517,Z 13,A -3.1198,B 0,C 0,E1 0.1598,E2 90.0713} C_DIS
LIN {X -6.3164,Y -1.9832,Z 13,A -3.1008,B 0,C 0,E1 0.1598,E2 90.0713} C_DIS
LIN {X -6.4918,Y -1.2906,Z 13,A -3.078,B 0,C 0,E1 0.1598,E2 90.0713} C_DIS
LIN {X -6.594,Y -0.5835,Z 13,A -3.052,B 0,C 0,E1 0.1598,E2 90.0713} C_DIS
LIN {X -6.6167,Y 0.1305,Z 13,A -3.0227,B 0,C 0,E1 0.1598,E2 90.0713} C_DIS
LIN {X -6.5661,Y 0.8431,Z 13,A -2.9908,B 0,C 0,E1 0.1598,E2 90.0713} C_DIS
LIN {X -6.4375,Y 1.546,Z 13,A -2.9565,B 0,C 0,E1 0.1598,E2 90.0713} C_DIS
LIN {X -6.2336,Y 2.2309,Z 13,A -2.9201,B 0,C 0,E1 0.1598,E2 90.0714} C_DIS
LIN {X -5.9583,Y 2.8903,Z 13,A -2.8822,B 0,C 0,E1 0.1598,E2 90.0715} C_DIS
LIN {X -5.6117,Y 3.5151,Z 13,A -2.8432,B 0,C 0,E1 0.1598,E2 90.0715} C_DIS
LIN {X -5.1989,Y 4.0983,Z 13,A -2.8034,B 0,C 0,E1 0.1598,E2 90.0717} C_DIS
Enddeposition()
END
